		FB_ModbusRead_PowerCol		: ARRAY[1.. CstNbPowerCol_PCS_G] OF FB_ModbusRead;
		FB_ModbusRead_DU			: ARRAY[1..CstNb_DU_G] OF FB_ModbusRead;
		FB_ModbusRead	          	: ARRAY[1..6] OF FB_ModbusRead; // (NA) FB for Modbus Reading
		FB_ModbusWrite				: ARRAY[1..7]  OF FB_ModbusWrite;
		AX_ModbusReadAlarmPowerCol	: ARRAY[1.. CstNbPowerCol_PCS_G] OF BOOL;
		AX_ModbusReadAlarmDU		: ARRAY[1.. CstNb_DU_G] OF BOOL;
		AX_ModbusReadAlarm			: ARRAY[1..6] OF BOOL;
		AX_ModbusReadAlarmId		: ARRAY[1..11] OF UDINT;
		AX_ModbusReadAlarmIdPowerCol: ARRAY[1.. CstNbPowerCol_PCS_G] OF UDINT;	
		AX_ModbusReadAlarmId_DU		: ARRAY[1.. CstNb_DU_G] OF UDINT;	
		AX_ModbusWriteAlarm			: ARRAY[1..7]  OF BOOL;
		AX_ModbusWriteAlarmId		: ARRAY[1..7]  OF UDINT;	
	
		MesBlock_Temp_1 			: ARRAY [1..120] OF WORD ; 		// (NA) Temporary Block with multiple modbus reading 
		MesBlock_Temp_2 			: ARRAY [0..120] OF WORD ; 		// (NA) Temporary Block with multiple modbus reading 
		MesBlock_Temp_3 			: ARRAY [1..120] OF WORD ; 		// (NA) Temporary Block with multiple modbus reading 
		MesBlock_Temp_4 			: ARRAY [1..120] OF WORD ; 		// (NA) Temporary Block with multiple modbus reading 
		MesBlock_Temp_5 			: ARRAY[1..CstNbPowerCol_PCS_G] OF ARRAY [1..32] OF WORD; 	// (NA) Temporary Block with multiple modbus reading 
		MesBlock_Temp_6 			: ARRAY[1..CstNb_DU_G] OF ARRAY [1..6] OF WORD ; 				// (NA) Temporary Block with multiple modbus reading 
		MesBlockWrite1_Temp 		: WORD;							// (NA) Temporary Block with multiple modbus writing (Caution : Double Word variables)
		MesBlockWrite2_Temp			: ARRAY[1..3] OF WORD;			// (NA) Temporary Block with multiple modbus writing (Caution : Double Word variables)
		MesBlockWrite3_Temp			: WORD;							// (NA) Temporary Block with multiple modbus writing (Caution : Double Word variables)
		MesBlockWrite4_Temp			: ARRAY[1..10] OF WORD;			// (NA) Temporary Block with multiple modbus writing (Caution : Double Word variables)
		MesBlockWrite5_Temp			: ARRAY[1..2] OF WORD;
		MesBlockWrite6_Temp			: WORD;
		MesBlockWrite7_Temp			: ARRAY[1..2] OF WORD;
		MesBlockWrite8_Temp			: WORD;

		TON_BJ						: ARRAY[1..10] OF TON; 


		AX_ADR_MB_Write				: ARRAY[1..2] OF  WORD := [100, 557];		// [40553, 40558, 40551];
		AX_QTY_MB_Write				: ARRAY[1..2] OF  BYTE := [1, 	1];                    // [1, 1, 1];
		                    		
		InvSetptP_temp				: REAL;
		InvSetptQ_temp				: REAL;
                            		
                            		
		AX_QTY_MB					: ARRAY[1..8] OF WORD := [120, 	120, 	10, 	1, 		5, 		120, 	120, 	50];
		AX_ADR_MB					: ARRAY[1..8] OF WORD := [1000, 1119, 	550, 	1391, 	5000, 	0000, 	5803, 	1350]; 			
		
	// M_STARTSTOP//
		StartStop_RTrig				: R_Trig;
              	
	// M_CP
		CalCP_CMD_StartStop			: BOOL; 						// Write command start;
		
		bTestComAlarm : BOOL;
		bTestComWarning : BOOL;
END_VAR

METHOD M_AlarmManagement
//////////////////
// Manages IntelliGen Alarms
/////////////////

VAR 
	// Method local variables (reinitialized at each cycle) 
	FB_AlarmCodeManager : FB_AlarmCodeManager ; 
	KK				: BYTE;		// For Loop 
	bComError		: BOOL := TRUE;
	bComWarning 	: BOOL;

	AX_BJHS			: ARRAY[1..10] OF BOOL;
END_VAR

bComError := (AX_ModbusReadAlarmPowerCol[1] AND AX_ModbusReadAlarmPowerCol[2] AND AX_ModbusReadAlarmPowerCol[3] AND AX_ModbusReadAlarmPowerCol[4] AND AX_ModbusReadAlarmPowerCol[5] AND AX_ModbusReadAlarmPowerCol[6]
		AND AX_ModbusReadAlarm[1] AND AX_ModbusReadAlarm[2] AND AX_ModbusReadAlarm[3] AND AX_ModbusReadAlarm[4]
		AND AX_ModbusWriteAlarm[1] AND AX_ModbusWriteAlarm[2]) OR bTestComAlarm;

bComWarning:= AX_ModbusReadAlarmPowerCol[1] OR AX_ModbusReadAlarmPowerCol[2] OR AX_ModbusReadAlarmPowerCol[3] OR AX_ModbusReadAlarmPowerCol[4] OR AX_ModbusReadAlarmPowerCol[5] OR AX_ModbusReadAlarmPowerCol[6]
		OR AX_ModbusReadAlarm[1] OR AX_ModbusReadAlarm[2] OR AX_ModbusReadAlarm[3] OR AX_ModbusReadAlarm[4]
		OR AX_ModbusWriteAlarm[1] OR AX_ModbusWriteAlarm[2] or bTestComWarning;


TON_ComAlarm(IN := bComError, PT := T#30S,Q=> MesDataExd.MesData.MesAlarmCom);
TON_ComWarning(IN := bComWarning, PT := T#30S, Q=> MesWarningCom);

// ALARM CODE //
	FB_AlarmCodeManager(
		bAlarm1			:= NOT MesDataExd.MesStateCom,							// INV Not Communicating
		bAlarm2			:= FALSE,												// 	
		bAlarm3			:= NOT MesDataExd.MesStateCBac,							// INV AC CB opened 
		bAlarm4			:= FALSE,												// 	
		bAlarm5			:= NOT MesDataExd.MesStateCBdc,							// INV DC CB opened 
		bAlarm6			:= FALSE,												// 
		bAlarm7			:= MesDataExd.MesFaultGnd,								// INV Ground Fault	
		bAlarm8			:= FALSE,												// 
		bAlarm9			:= NOT MesDataExd.MesStateNoAlert, 						// INV ID = 9, inverter has detected an abnormal fault which prevents operation
		bAlarm10		:= FALSE, //
		bAlarm11		:= FALSE, //
		bAlarm12		:= FALSE, //
		bAlarm13		:= FALSE, //
		bAlarm14		:= FALSE, //
		bAlarm15		:= MesDataExd.MesData.MesAlarmCom, 						 // No communication frames for the past 30 seconds 					 			#COM
		wAlarmCode		=> MesDataExd.MesData.MesAlarmCode);					

// WARNING CODE //
	FB_AlarmCodeManager(
 		bAlarm1			:= MesWarningCom, 										// A frame failed for the last 30s 												#COM
		bAlarm2			:= FALSE, //
		bAlarm3			:= NOT MesDataExd.Mesdata.MesCP_Read, 	  							// No permission to read from SCADA
		bAlarm4			:= MesDataExd.ParamID_PMode <> 0,						// INV active power setpoint is not MPPT  										#Equipment
		bAlarm5			:= NOT MesDataExd.Mesdata.MesCP_Write,								// No permission to write from SCADA							
		bAlarm6			:= FALSE, //
		bAlarm7			:= FALSE, //
		bAlarm8			:= FALSE,												//
		bAlarm9			:= IN_SetptPlimit_Local < ParamPn,  	// INV local active power setpoint is under nominal active power 
		bAlarm10		:= NOT RS_StartStop_Local.Q1,       					// Local Stop Command 
		bAlarm11		:= FALSE,						 						// 
		bAlarm12		:= FALSE, 												//
		bAlarm13		:= FALSE,												// 
		bAlarm14		:= FALSE,												// 
		bAlarm15		:= FALSE, 												//
		wAlarmCode		=> MesDataExd.MesData.MesWarningCode);	
// EVENT CODE //
	FB_AlarmCodeManager(
		bAlarm1			:= FALSE, //
		bAlarm2			:= FALSE, //
		bAlarm3			:= FALSE, //
		bAlarm4			:= FALSE, //
		bAlarm5			:= FALSE, //
		bAlarm6			:= FALSE, //
		bAlarm7			:= MesDataExd.MesData.MesState_INV = 24,  				// Econmode: activated the econmode to save MV losses
		bAlarm8			:= MesDataExd.MesData.MesState_INV = 23,  				// Autonight: switches to autonight state
		bAlarm9			:= MesDataExd.MesData.MesState_INV = 20,  				// Premagnetization: MV transformer pre-mag
		bAlarm10		:= MesDataExd.MesData.MesState_INV = 19,  				// Filter contactors: LC filter contact activated
		bAlarm11		:= NOT RS_StartStop.Q1, 								// Stop command for INV 
		bAlarm12		:= MesDataExd.MesData.MesState_INV = 0,  				// Power Up
		bAlarm13		:= MesDataExd.MesData.MesState_INV = 1,  				// Init: basic condition are being checked
		bAlarm14		:= MesDataExd.MesData.MesState_INV = 2,  				// Off: stopped
		bAlarm15		:= MesDataExd.MesData.MesState_INV = 3,  				// PCHG : Precharge
		wAlarmCode		=>  MesDataExd.MesData.MesEventCode);
// EVENT CODE //
	FB_AlarmCodeManager(
		bAlarm1			:= MesDataExd.MesData.MesState_INV = 4,  				// REA : Ready, wainting for start command
		bAlarm2			:= MesDataExd.MesData.MesState_INV = 5,  				// WAIT: Waiting for delay time
		bAlarm3			:= MesDataExd.MesData.MesState_INV = 6,  				// ON: inverter operting normally
		bAlarm4			:= MesDataExd.MesData.MesState_INV = 7,  				// Stop: inverter is stopping
		bAlarm5			:= MesDataExd.MesData.MesState_INV = 8,  				// Discharge: capacitor discharging for 1min
		bAlarm6			:= MesDataExd.MesData.MesState_INV = 9,  				// Fault: check fault code
		bAlarm7			:= MesDataExd.MesData.MesState_INV = 10,  				// LVRT: low voltage ride through
		bAlarm8			:= MesDataExd.MesData.MesState_INV = 11,  				// OVRT: Over voltage ride through
		bAlarm9			:= MesDataExd.MesData.MesState_INV = 12,  				// NGHT: Night
		bAlarm10		:= MesDataExd.MesData.MesState_INV = 13,  				// NDCO: Night DC off: DC opened, no heating or night mode
		bAlarm11		:= MesDataExd.MesData.MesState_INV = 14,  				// Standby: waiting for conditions to perform softcharge
		bAlarm12		:= MesDataExd.MesData.MesState_INV = 15,  				// HVPL: high voltage phase lost
		bAlarm13		:= MesDataExd.MesData.MesState_INV = 16,  				// Trackers: trackers mode running
		bAlarm14		:= MesDataExd.MesData.MesState_INV = 17,  				// Pre-on: soft charge and synchronization
		bAlarm15		:= MesDataExd.MesData.MesState_INV = 18,  				// Diagnosis: extended self-diagnosis									
		wAlarmCode		=>  MesDataExd.MesEventCode2);

				
(*
	FB_AlarmCodeManager(
		bAlarm0			:= FALSE, 			// P Curtail -  no curtail
		bAlarm1			:= FALSE, 			// P Curtail -  Id : Current close loop
		bAlarm2			:= FALSE, 			// P Curtail -  P : Power close loop
		bAlarm3			:= FALSE, 			// P Curtail -  Vdc : voltage close loop
		bAlarm4			:= FALSE, 			// P Curtail -  HT
		bAlarm5			:= FALSE, 			// P Curtail -  STAT
		bAlarm6			:= FALSE, 			// P Curtail -  R
		bAlarm7			:= FALSE, 			// P Curtail -  Night : voltage dc night
		bAlarm8			:= FALSE, 			// 
		bAlarm9			:= FALSE, 			// 
		bAlarm10		:= FALSE, 			// 
		bAlarm11		:= FALSE,			// 
		bAlarm12		:= FALSE,			// 
		bAlarm13		:= FALSE,			// 
		bAlarm14		:= FALSE,			// 
		bAlarm15		:= FALSE,			// 		
		wAlarmCode		=>  MesDataExd.MesStatusCurtail_P);

	FB_AlarmCodeManager(
		bAlarm0			:= FALSE, 			// Q Curtail - CosPhi
		bAlarm1			:= FALSE, 			// Q Curtail - Iq : Current close loop
		bAlarm2			:= FALSE, 			// Q Curtail - Q : Power cose loop
		bAlarm3			:= FALSE, 			// Q Curtail - QV : QV Curve
		bAlarm4			:= FALSE, 			// Q Curtail - HT
		bAlarm5			:= FALSE, 			// Q Curtail - R
		bAlarm6			:= FALSE, 			// 
		bAlarm7			:= FALSE, 			// 
		bAlarm8			:= FALSE, 			// 
		bAlarm9			:= FALSE, 			// 
		bAlarm10		:= FALSE, 			// 
		bAlarm11		:= FALSE,			// 
		bAlarm12		:= FALSE,			// 
		bAlarm13		:= FALSE,			// 
		bAlarm14		:= FALSE,			// 
		bAlarm15		:= FALSE,			// 		
		wAlarmCode		=>  MesDataExd.MesStatusCurtail_Q);

	FB_AlarmCodeManager(
		bAlarm0			:= FALSE, 			// State - Stopped
		bAlarm1			:= FALSE, 			// State - MPPT
		bAlarm2			:= FALSE, 			// State - Sleeping
		bAlarm3			:= FALSE, 			// State - Starting
		bAlarm4			:= FALSE, 			// State - Throttled
		bAlarm5			:= FALSE, 			// State - Shutting Down
		bAlarm6			:= FALSE, 			// State - Fault
		bAlarm7			:= FALSE, 			// State - Standby
		bAlarm8			:= FALSE, 			// 
		bAlarm9			:= FALSE, 			// 
		bAlarm10		:= FALSE, 			// 
		bAlarm11		:= FALSE,			// 
		bAlarm12		:= FALSE,			// 
		bAlarm13		:= FALSE,			// 
		bAlarm14		:= FALSE,			// 
		bAlarm15		:= FALSE,			// 		
		wAlarmCode		=>  MesDataExd.MesData.MesState);		
		
		
*)				
FOR KK := 1 TO CstNbPowerCol_PCS_G DO
	FB_AlarmCodeManager(
		bAlarm1			:= MesDataExd.AX_PowerCol[KK].MesState_Inv = 22, 			// 22, Idle: Module waits 5s before starting
		bAlarm2			:= MesDataExd.AX_PowerCol[KK].MesState_Inv = 1, 			// 1, Stop: Module is stopped
		bAlarm3			:= MesDataExd.AX_PowerCol[KK].MesState_Inv = 2, 			// 2, Softcharge: Module performing softcharge
		bAlarm4			:= MesDataExd.AX_PowerCol[KK].MesState_Inv = 3, 			// 3, Ready: waiting for start command
		bAlarm5			:= MesDataExd.AX_PowerCol[KK].MesState_Inv = 4, 			// 4, LCL: LCL filter contact activated
		bAlarm6			:= MesDataExd.AX_PowerCol[KK].MesState_Inv = 5, 			// 5, Main AC: main contact activated, waiting feedback
		bAlarm7			:= MesDataExd.AX_PowerCol[KK].MesState_Inv = 6, 			// 6, Main AC Wait: module waits 100ms with ac contact closed
		bAlarm8			:= MesDataExd.AX_PowerCol[KK].MesState_Inv = 7, 			// 7, Run: Module injecting
		bAlarm9			:= MesDataExd.AX_PowerCol[KK].MesState_Inv = 8, 			// 8, nMain AC: AC open, LCL contactor closed during 100ms
		bAlarm10		:= MesDataExd.AX_PowerCol[KK].MesState_Inv = 9, 			// 9, Discharge: Module performing active discharge
		bAlarm11		:= MesDataExd.AX_PowerCol[KK].MesState_Inv = 10,			// 10, VRT event occured in network
		bAlarm12		:= MesDataExd.AX_PowerCol[KK].MesState_Inv = 11,			// 11, Trackers mode
		bAlarm13		:= MesDataExd.AX_PowerCol[KK].MesState_Inv = 14,			// 14, Fault AC overcurrent
		bAlarm14		:= MesDataExd.AX_PowerCol[KK].MesState_Inv = 15,			// 15, Fault overvoltage
		bAlarm15		:= MesDataExd.AX_PowerCol[KK].MesState_Inv = 17,			// 17, Fault exit OV wait
		wAlarmCode		=>  MesDataExd.AX_PowerCol[KK].MesState_Inv_ID);	
		
		
	FB_AlarmCodeManager(
		bAlarm1			:= MesDataExd.AX_PowerCol[KK].MesState_Inv = 55, 			// 55,  Init : Module is initializing
		bAlarm2			:= MesDataExd.AX_PowerCol[KK].MesState_Inv = 18, 			// 18, Fault exit wait
		bAlarm3			:= MesDataExd.AX_PowerCol[KK].MesState_Inv = 19, 			// 19, Softcharge fault
		bAlarm4			:= MesDataExd.AX_PowerCol[KK].MesState_Inv = 20, 			// 20, Fault
		bAlarm5			:= MesDataExd.AX_PowerCol[KK].MesState_Inv = 116, 			// 116, Module disabled SC: softcharge fault
		bAlarm6			:= MesDataExd.AX_PowerCol[KK].MesState_Inv = 159, 			// 159, Master FPGA comms error
		bAlarm7			:= FALSE, //
		bAlarm8			:= FALSE, //
		bAlarm9			:= FALSE, //
		bAlarm10		:= FALSE, //
		bAlarm11		:= FALSE, //
		bAlarm12		:= FALSE, //
		bAlarm13		:= FALSE, //
		bAlarm14		:= FALSE, //
		bAlarm15		:= FALSE, //
		wAlarmCode		=>  MesDataExd.AX_PowerCol[KK].MesState_Inv_ID2);	
END_FOR
END_METHOD

METHOD M_CP
//////////////////
//  Emulator
/////////////////

VAR 
	// Method local variables (reinitialized at each cycle) 
	
END_VAR

	
SUPER^.M_CP();
CalCP_CMD_StartStop	:= FB_ModbusRead[1].OUT_NbRead > 0 AND SEL(MesDataExd.MesStartDisabled, TRUE, NOT RS_StartStop.Q1); // FB_ModbusRead[1].OUT_NbRead > 0 AND (MesDataExd.MesStartDisabled  <> NOT  RS_StartStop.Q1);  




Trig_Cmd_Read(CLK:=IN_CmdToggleRead);
Trig_Cmd_Write(CLK:=IN_CmdToggleWrite);
	
IF Trig_Cmd_Read.Q THEN
	IN_CmdToggleRead := FALSE;
	MesDataExd.MesData.MesCP_Read := NOT MesDataExd.MesData.MesCP_Read;
END_IF


IF Trig_Cmd_Write.Q THEN
	IN_CmdToggleWrite := FALSE;
	MesDataExd.MesData.MesCP_Write := NOT MesDataExd.MesData.MesCP_Write;
END_IF
END_METHOD

{attribute 'object_name' := 'M_Curtail'}
METHOD M_Curtail
//////////////////
// Write Curtail Command through modbus to PV inverters.  
//////////////////
VAR 
	// Method local variables (reinitialized at each cycle) 

	MW					: FB_MergeWordsToFloat;
	MW_1				: FB_SplitFloatToWords;

	KK: INT;
END_VAR
SUPER^.M_Curtail() ; 

// MODBUS VARIABLE FORMATING //
// Setpoints //

IF IN_SetptPlimit = 0 AND (MesDataExd.MesData.MesState.0 OR MesDataExd.MesData.MesState.2 OR MesDataExd.MesData.MesState.3) THEN
	IN_SetptPlimit := 100;
END_IF

IF MesDataExd.OUT_CmdInvLocal THEN
	InvSetptP_temp	:= 100*MIN(100, 100 * IN_SetptPlimit_Local / ParamPn); 
	InvSetptQ_temp	:= 100*MIN(100, 100 * IN_SetptQ_Local / ParamQn); 

	MesDataExd.MesData.OUT_SetptPLimit :=  IN_SetptPlimit_Local; 
	MesDataExd.MesData.OUT_SetptQ :=  IN_SetptQ_Local; 	

ELSE
	InvSetptP_temp	:= 10000*IN_SetptPlimit / ParamPn; 
	InvSetptQ_temp	:= 10000*IN_SetptQ / ParamQn; 

	MesDataExd.MesData.OUT_SetptPLimit :=  IN_SetptPlimit; 
	MesDataExd.MesData.OUT_SetptQ :=  IN_SetptQ; 
	
END_IF	

		
	
	MesBlockWrite4_Temp[1] := REAL_TO_WORD(InvSetptP_temp);
	MesBlockWrite4_Temp[2] := REAL_TO_WORD(InvSetptQ_temp);
			
		
		FB_ModbusWrite[1]
	(
		pSrcAddr := ADR (MesBlockWrite4_Temp[1]),
		sIPAddr := ParamIPAddress,
		tTimeout := ParamTimeout,
		nMBAddr := AX_ADR_MB_Write[1],
		nTCPport := ParamTCPPort,
		cbLength := SIZEOF(MesBlockWrite4_Temp[1]),
		nQuantity := AX_QTY_MB_Write[1],
		nUnitID := ParamUnitID,
		WriteCmd := ClockWrite AND MesDataExd.Mesdata.MesCP_Write  ,
		Reset := CmdClearFault_G OR IN_CmdReset_L,
		ErrorId => AX_ModbusWriteAlarmId[1],
		ModbusWriteAlarm => AX_ModbusWriteAlarm[1]
	);

	FB_ModbusWrite[2]
(
	pSrcAddr := ADR (MesBlockWrite4_Temp[2]),
	sIPAddr := ParamIPAddress,
	tTimeout := ParamTimeout,
	nMBAddr := AX_ADR_MB_Write[2],
	nTCPport := ParamTCPPort,
	cbLength := SIZEOF(MesBlockWrite4_Temp[2]),
	nQuantity := AX_QTY_MB_Write[2],
	nUnitID := ParamUnitID,
	WriteCmd := ClockWrite AND MesDataExd.Mesdata.MesCP_Write  ,
	Reset := CmdClearFault_G OR IN_CmdReset_L,
	ErrorId => AX_ModbusWriteAlarmId[2],
	ModbusWriteAlarm => AX_ModbusWriteAlarm[2]
);
END_METHOD

METHOD M_Evaluate
VAR_INPUT
END_VAR
IN_SetptPlimit 	:= IN_SetptPlimit;
IN_SetptQ		:= IN_SetptQ;
END_METHOD

METHOD M_Execute
//////////////////
//  Method Calls 
/////////////////

VAR 
	// Method local variables (reinitialized at each cycle) 

END_VAR
IF  bInit THEN
	M_Init();
	bInit:= FALSE ; 
ELSIF CmdInit_G THEN 
	bInit:= TRUE ;
END_IF

SUPER^.M_Execute(); 

//M_Evaluate();
M_AlarmManagement();
END_METHOD

METHOD M_Init

VAR
	bCompleted 			: BOOL := FALSE;
	AX_ADR_MB			: WORD := 44253; 
END_VAR
ParamPn := 3800;
IN_SetptPlimit_Local := 3800;

// Watchdog timer start
Watchdog_CP_Write := TRUE;
ParamClockReadTime := T#1S;
ParamClockWriteTime := T#200MS;
END_METHOD

{attribute 'object_name' := 'M_Read'}
METHOD M_Read
//////////
// Read Method for PE SKID HEMK : Modbus reading
//////////
VAR
	// Method local variables (reinitialized at each cycle) 
	MW_Float			: FB_MergeWordsToFloat;
	MW_REAL				: FB_MergeWordsToDint;
	MW_UInt				: FB_MergeWordsToUint;
	
	
	EacInj_Interm1		: ULINT;
	EacCon_Interm1		: ULINT;
	EreacCapa_Interm1	: ULINT;
	EreacInd_Interm1	: ULINT;
	EacInj_Day_Interm1	: ULINT;
	
	EacInj_Interm2		: ULINT;
	EacCon_Interm2		: ULINT;
	EreacCapa_Interm2	: ULINT;
	EreacInd_Interm2	: ULINT;
	EacInj_Day_Interm2	: ULINT;
	
	Temp_Cells_Transfo	: WORD;
	Temp_Cells_Transfo_2: WORD;
	Temp_Cells_Transfo_3: WORD;
	Temp_Cells_Transfo_4: WORD;
	MesResistor			: REAL;
	
	KK					: BYTE;						 // Index to loop over modbus blocks 	
	JJ					: BYTE;
END_VAR
IF MesDataExd.MesData.MesCP_Read THEN		

// MODBUS REQUEST//
	//Electrical Measurements + Ground Measurements
	FB_ModbusRead[1]
	(
		nTCPPort		:= ParamTcpPort,
		ClockRead		:= MesDataExd.Mesdata.MesCP_Read AND ClockRead, 
		Reset			:= CmdClearFault_G OR IN_CmdReset_L,
		sIPAddr			:=ParamIPAddress ,
		nUnitID			:= 1, 
		tTimeout		:= ParamTimeout,
		nQuantity		:= AX_QTY_MB[1] , 
		nMBAddr			:= AX_ADR_MB[1] , 
		cbLength		:= SIZEOF(MesBlock_Temp_1) , 
		pDestAddr		:= ADR(MesBlock_Temp_1) , 
		ModbusReadAlarm	=>AX_ModbusReadAlarm[1] , 
		ErrorId			=> AX_ModbusReadAlarmId[1]
	);
		
	//Production Measurements
	FB_ModbusRead[2]
	(
		nTCPPort		:= ParamTcpPort,
		ClockRead		:= MesDataExd.Mesdata.MesCP_Read AND ClockRead, 
		Reset			:= CmdClearFault_G OR IN_CmdReset_L,
		sIPAddr			:=ParamIPAddress , 
		nUnitID			:= 1, 
		tTimeout		:= ParamTimeout,
		nQuantity		:= AX_QTY_MB[2] , 
		nMBAddr			:= AX_ADR_MB[2] , 
		cbLength		:= SIZEOF(MesBlock_Temp_2) , 
		pDestAddr		:= ADR(MesBlock_Temp_2) , 
		ModbusReadAlarm	=>AX_ModbusReadAlarm[2] , 
		ErrorId			=> AX_ModbusReadAlarmId[2]
	);
	
	// Status Summary + Event Summary
	FB_ModbusRead[3]
	(
		nTCPPort		:= ParamTcpPort,
		ClockRead		:= MesDataExd.MesData.MesCP_Read AND ClockRead, 
		Reset			:= CmdClearFault_G OR IN_CmdReset_L,
		sIPAddr			:=ParamIPAddress , 
		nUnitID			:= 1, 
		tTimeout		:= ParamTimeout,
		nQuantity		:= AX_QTY_MB[3] , 
		nMBAddr			:= AX_ADR_MB[3] , 
		cbLength		:= SIZEOF(MesBlock_Temp_3) , 
		pDestAddr		:= ADR(MesBlock_Temp_3) , 
		ModbusReadAlarm	=>AX_ModbusReadAlarm[3] , 
		ErrorId			=> AX_ModbusReadAlarmId[3]
	);
	
	//Number running modules
	FB_ModbusRead[4]
	(
		nTCPPort		:= ParamTcpPort,
		ClockRead		:= MesDataExd.MesData.MesCP_Read AND ClockRead, 
		Reset			:= CmdClearFault_G OR IN_CmdReset_L,
		sIPAddr			:= ParamIPAddress , 
		nUnitID			:= 1, 
		tTimeout		:= ParamTimeout,
		nQuantity		:= AX_QTY_MB[4], 
		nMBAddr			:= AX_ADR_MB[4], 
		cbLength		:= SIZEOF(MesBlock_Temp_4), 
		pDestAddr		:= ADR(MesBlock_Temp_4), 
		ModbusReadAlarm	=> AX_ModbusReadAlarm[4], 
		ErrorId			=> AX_ModbusReadAlarmId[4]
	);
	
	//Power Commands
	FOR KK:= 1 TO  CstNbPowerCol_PCS_G DO 
		FB_ModbusRead_PowerCol[KK]
		(
				nTCPPort		:= ParamTcpPort,
				ClockRead		:= MesDataExd.Mesdata.MesCP_Read AND ClockRead, 
				Reset			:= CmdClearFault_G OR IN_CmdReset_L,
				sIPAddr			:=ParamIPAddress , 
				nUnitID			:= 1, 
				tTimeout		:= ParamTimeout,
				nQuantity		:= 32 , 
				nMBAddr			:= 5000 + 32*(KK-1) ,  
				cbLength		:= SIZEOF(MesBlock_Temp_5[KK]) , 
				pDestAddr		:= ADR(MesBlock_Temp_5[KK]) , 
				ModbusReadAlarm	=>AX_ModbusReadAlarmPowerCol[KK] , 
				ErrorId			=> AX_ModbusReadAlarmIdPowerCol[KK]
		);
	END_FOR
		
	FOR KK:= 1 TO  CstNb_DU_G DO 
		FB_ModbusRead_DU[KK]
		(
				nTCPPort		:= ParamTcpPort,
				ClockRead		:= MesDataExd.Mesdata.MesCP_Read AND ClockRead, 
				Reset			:= CmdClearFault_G OR IN_CmdReset_L,
				sIPAddr			:= ParamIPAddress , 
				nUnitID			:= 1, 
				tTimeout		:= ParamTimeout,
				nQuantity		:= 6, 
				nMBAddr			:= 5800 + 6*(KK-1),  
				cbLength		:= SIZEOF(MesBlock_Temp_6[KK]), 
				pDestAddr		:= ADR(MesBlock_Temp_6[KK]), 
				ModbusReadAlarm	=>AX_ModbusReadAlarmDU[KK], 
				ErrorId			=> AX_ModbusReadAlarmId_DU[KK]
		);
	END_FOR
      

    MW_REAL(WORD_STRONG:= MesBlock_Temp_1[  1], SIGNED:=FALSE, FIX:=0 , SIZE:=1, VAR_OUT:=MesDataExd.MesU12);
	MW_REAL(WORD_STRONG:= MesBlock_Temp_1[  2], SIGNED:=FALSE, FIX:=0 , SIZE:=1, VAR_OUT:=MesDataExd.MesU23);
	MW_REAL(WORD_STRONG:= MesBlock_Temp_1[  3], SIGNED:=FALSE, FIX:=0 , SIZE:=1, VAR_OUT:=MesDataExd.MesU31);
	MW_REAL(WORD_STRONG:= MesBlock_Temp_1[  4], SIGNED:=FALSE, FIX:=1 , SIZE:=1, VAR_OUT:=MesDataExd.MesI1);
	MW_REAL(WORD_STRONG:= MesBlock_Temp_1[  5], SIGNED:=FALSE, FIX:=1 , SIZE:=1, VAR_OUT:=MesDataExd.MesI2);
	MW_REAL(WORD_STRONG:= MesBlock_Temp_1[  6], SIGNED:=FALSE, FIX:=1 , SIZE:=1, VAR_OUT:=MesDataExd.MesI3);
	MW_REAL(WORD_STRONG:= MesBlock_Temp_1[  8], SIGNED:=TRUE, FIX:=0 , SIZE:=1, VAR_OUT:=MesDataExd.MesData.MesP);
	MW_REAL(WORD_STRONG:= MesBlock_Temp_1[  9], SIGNED:=TRUE, FIX:=0 , SIZE:=1, VAR_OUT:=MesDataExd.MesData.MesQ);
	MW_REAL(WORD_STRONG:= MesBlock_Temp_1[ 10], SIGNED:=FALSE, FIX:=0 , SIZE:=1, VAR_OUT:=MesDataExd.MesData.MesS);
	MW_REAL(WORD_STRONG:= MesBlock_Temp_1[ 11], SIGNED:=TRUE, FIX:=3 , SIZE:=1, VAR_OUT:=MesDataExd.MesData.MesCosPhi);
	MW_REAL(WORD_STRONG:= MesBlock_Temp_1[ 12], SIGNED:=FALSE, FIX:=2 , SIZE:=1, VAR_OUT:=MesDataExd.MesData.MesFreq);
	MW_REAL(WORD_STRONG:= MesBlock_Temp_1[ 52], SIGNED:=FALSE, FIX:=0 , SIZE:=1, VAR_OUT:=MesDataExd.MesData.MesUdc);  
	MW_REAL(WORD_STRONG:= MesBlock_Temp_1[ 61], SIGNED:=FALSE, FIX:=0 , SIZE:=1, VAR_OUT:=MesDataExd.MesData.MesPdc);
	MW_REAL(WORD_STRONG:= MesBlock_Temp_1[ 62], SIGNED:=FALSE, FIX:=0 , SIZE:=1, VAR_OUT:=MesDataExd.MesData.MesIdc); 
	MW_REAL(WORD_STRONG:= MesBlock_Temp_1[ 104], Word_WEAK:= MesBlock_Temp_1[105], SIGNED:=FALSE, FIX:=3 , SIZE:=2, VAR_OUT:=MesDataExd.MesData.MesInsuResistor);
	MW_REAL(WORD_STRONG:= MesBlock_Temp_1[ 114], Word_WEAK:= MesBlock_Temp_1[115], SIGNED:=FALSE, FIX:=0 , SIZE:=2, VAR_OUT:=MesDataExd.MesInsuResistor_AC);
	

	
	
// INV status
	MW_REAL(WORD_STRONG:= MesBlock_Temp_2[ 0], SIGNED:=FALSE, FIX:=0 , SIZE:=1, VAR_OUT:=MesDataExd.MesTemp_DU);
	MW_UInt(WORD_STRONG:= MesBlock_Temp_2[ 1], VAR_OUT := MesDataExd.MesAlarm_Control); 	
	MW_UInt(WORD_STRONG:= MesBlock_Temp_2[ 2], VAR_OUT := MesDataExd.MesWarning_Control); 	
	MW_UInt(WORD_STRONG:= MesBlock_Temp_2[ 3], VAR_OUT := MesDataExd.MesData.MesState_INV); 	
	MW_REAL(WORD_STRONG:= MesBlock_Temp_2[ 4], SIGNED:=FALSE, FIX:=0 , SIZE:=1, VAR_OUT:=MesDataExd.MesTemp_Control);
	MW_REAL(WORD_STRONG:= MesBlock_Temp_2[ 5], SIGNED:=FALSE, FIX:=0 , SIZE:=1, VAR_OUT:=MesDataExd.MesTemp_IGBTmax);
	MW_REAL(WORD_STRONG:= MesBlock_Temp_2[ 6], SIGNED:=FALSE, FIX:=0 , SIZE:=1, VAR_OUT:=MesDataExd.MesTemp_PowerColmax);	

	MW_REAL(WORD_STRONG:= MesBlock_Temp_2[21], SIGNED:=FALSE, FIX:=4, SIZE:=1, VAR_OUT:=MesDataExd.MesSetptP);
	MW_REAL(WORD_STRONG:= MesBlock_Temp_2[22], SIGNED:=FALSE, FIX:=4, SIZE:=1, VAR_OUT:=MesDataExd.MesSetptQ);
	MesDataExd.MesCP_Start := WORD_TO_BOOL(MesBlock_Temp_2[ 31]);
	
// Power column/module variables
		MesDataExd.MesStatusCurtail_P := MesBlock_Temp_3[1]; 
		MesDataExd.MesStatusCurtail_Q := MesBlock_Temp_3[2]; 

	
		MesDataExd.MesNbRunningModules := WORD_TO_UINT(MesBlock_Temp_4[1]);
	
	FOR KK:= 1 TO CstNbPowerCol_PCS_G DO 	
		MW_UInt(WORD_STRONG:= MesBlock_Temp_5[KK][ 1], VAR_OUT := MesDataExd.AX_PowerCol[KK].MesState_Inv);
	
		MW_REAL(WORD_STRONG:= MesBlock_Temp_5[KK][ 2], SIGNED:=FALSE, FIX:=1 , SIZE:=1, VAR_OUT := MesDataExd.AX_PowerCol[KK].MesData.MesI1);
		MW_REAL(WORD_STRONG:= MesBlock_Temp_5[KK][ 3], SIGNED:=FALSE, FIX:=1 , SIZE:=1, VAR_OUT := MesDataExd.AX_PowerCol[KK].MesData.MesI2);
		MW_REAL(WORD_STRONG:= MesBlock_Temp_5[KK][ 4], SIGNED:=FALSE, FIX:=1 , SIZE:=1, VAR_OUT := MesDataExd.AX_PowerCol[KK].MesData.MesI3);
		MW_REAL(WORD_STRONG:= MesBlock_Temp_5[KK][ 5], SIGNED:=FALSE, FIX:=1 , SIZE:=1, VAR_OUT := MesDataExd.AX_PowerCol[KK].MesData.MesIdc);
		MW_REAL(WORD_STRONG:= MesBlock_Temp_5[KK][ 8], SIGNED:=FALSE, FIX:=0 , SIZE:=1, VAR_OUT := MesDataExd.AX_PowerCol[KK].MesData.MesUdc);
		MW_REAL(WORD_STRONG:= MesBlock_Temp_5[KK][ 9], SIGNED:=FALSE, FIX:=1 , SIZE:=1, VAR_OUT := MesDataExd.AX_PowerCol[KK].MesData.MesP);
		MW_REAL(WORD_STRONG:= MesBlock_Temp_5[KK][ 10], SIGNED:=FALSE, FIX:=1 , SIZE:=1, VAR_OUT:= MesDataExd.AX_PowerCol[KK].MesData.MesQ);
		MW_REAL(WORD_STRONG:= MesBlock_Temp_5[KK][ 11], SIGNED:=FALSE, FIX:=0 , SIZE:=1, VAR_OUT:= MesDataExd.AX_PowerCol[KK].MesTemp);
		MW_REAL(WORD_STRONG:= MesBlock_Temp_5[KK][ 12], SIGNED:=FALSE, FIX:=0 , SIZE:=1, VAR_OUT:= MesDataExd.AX_PowerCol[KK].MesTempmax);
		
		MesDataExd.AX_PowerCol[KK].MesStateIO := MesBlock_Temp_5[KK][13];
		MW_REAL(WORD_STRONG:= MesBlock_Temp_5[KK][ 32], SIGNED:=FALSE, FIX:=0 , SIZE:=1, VAR_OUT:=MesDataExd.AX_PowerCol[KK].MesHygro);
	END_FOR
		
	//// DU Channels ///////
	FOR KK:= 1 TO CstNb_DU_G DO 
	// Status
		MW_UInt(WORD_STRONG:= MesBlock_Temp_6[KK][4], VAR_OUT := MesDataExd.AX_DU[KK].MesIDState); 
			
	// Current
		MW_REAL(WORD_STRONG:= MesBlock_Temp_6[KK][5], SIGNED:=TRUE, FIX:=1, SIZE:=1, VAR_OUT := MesDataExd.AX_DU[KK].MesI); // dA ?
	
	// Voltage
		MW_REAL(WORD_STRONG:= MesBlock_Temp_6[kk][6], SIGNED:=TRUE, FIX:=1, SIZE:=1, VAR_OUT := MesDataExd.AX_DU[KK].MesU); // dV ?
				
	END_FOR
	// Evaluate 
	MesDataExd.MesData.MesI						:= (MesDataExd.MesI1 + MesDataExd.MesI2 + MesDataExd.MesI3) /3;
	MesDataExd.MesData.MesU						:= (MesDataExd.MesU12 + MesDataExd.MesU23 + MesdataExd.MesU31) /3 ; 
	                                			
	MesDataExd.MesData.MesAlarmCom  			:= TON_ComAlarm.Q; 
	MesDataExd.MesStateCom 						:= NOT MesDataExd.MesData.MesAlarmCom; 
	MesDataExd.MesData.MesTemp					:= MesDataExd.MesTemp_Control;                         			                                    	
END_IF
END_METHOD

METHOD M_StartStop
VAR
	KK : UINT;
	AX_ADR_MB			: ARRAY[1..3] OF WORD := [43010, 43200, 44252];
	AX_QTY_MB			: ARRAY[1..3] OF BYTE := [3, 1, 1];
END_VAR
SUPER^.M_StartStop(); 

// Start/Stop
Trig_Local_Start(CLK:=IN_CmdStart_Local);
Trig_Local_Stop(CLK:=IN_CmdStop_Local);

Trig_Start(CLK:=IN_CmdStart);
Trig_Stop(CLK:=IN_CmdStop);

IF Trig_Local_Start.Q OR Trig_Local_Stop.Q OR Trig_Stop.Q OR Trig_Start.Q THEN
	RS_StartStop(SET:=(IN_CmdStart_Local AND NOT IN_CmdStop_Local) OR (IN_CmdStart AND NOT (IN_CmdStop OR IN_CmdStop_Local)), 
			 Reset1 := IN_CmdStop_Local OR (IN_CmdStop AND NOT IN_CmdStart_Local)); 
END_IF

// Emergency stop 
Trig_Local_EmergencyStop(CLK:=IN_CmdEmergencyStop_Local);

// Reset 
Trig_Reset(CLK:= IN_CmdReset_L);

FB_ModbusWrite[5](WriteCmd := FALSE);
FB_ModbusWrite[6](WriteCmd := FALSE);
//FB_ModbusWrite[7](WriteCmd := FALSE);

// Start/Stop/Reset
MesBlockWrite2_Temp[1] := BOOL_TO_WORD(RS_StartStop.Q1);
MesBlockWrite2_Temp[2] := BOOL_TO_WORD(NOT RS_StartStop.Q1);
MesBlockWrite2_Temp[3] := BOOL_TO_WORD(Trig_Reset.Q);
// Emergency stop 
MesBlockWrite3_Temp    := BOOL_TO_WORD(Trig_Local_EmergencyStop.Q);

MesDataExd.MesData.OUT_CmdStart := RS_StartStop.Q1 ; 
MesDataExd.MesData.OUT_CmdStop  := NOT RS_StartStop.Q1 ; 	
MesDataExd.OUT_CmdReset			:= 	Trig_Reset.Q;
MesDataExd.OUT_CmdEmergencyStop := Trig_Local_EmergencyStop.Q;

StartStop_RTrig(CLK:=CalCP_CMD_StartStop);

	FB_ModbusWrite[5]
	(
		pSrcAddr := ADR (MesBlockWrite2_Temp),
		sIPAddr := ParamIPAddress,
		tTimeout := ParamTimeout,
		nMBAddr := AX_ADR_MB[1],
		nTCPport := ParamTCPPort,
		cbLength := SIZEOF(MesBlockWrite2_Temp),
		nQuantity := AX_QTY_MB[1],
		nUnitID := ParamUnitID,
		WriteCmd := StartStop_RTrig.Q AND MesDataExd.Mesdata.MesCP_Write ,
		Reset := CmdClearFault_G,
		ErrorId => AX_ModbusWriteAlarmId[5],
		ModbusWriteAlarm => AX_ModbusWriteAlarm[5]
	);

	FB_ModbusWrite[6]
	(
		pSrcAddr := ADR (MesBlockWrite3_Temp),
		sIPAddr := ParamIPAddress,
		tTimeout := ParamTimeout,
		nMBAddr := AX_ADR_MB[2],
		nTCPport := ParamTCPPort,
		cbLength := SIZEOF(MesBlockWrite3_Temp),
		nQuantity := AX_QTY_MB[2],
		nUnitID := ParamUnitID,
		WriteCmd := Trig_Local_EmergencyStop.Q AND MesDataExd.Mesdata.MesCP_Write,
		Reset := CmdClearFault_G,
		ErrorId => AX_ModbusWriteAlarmId[6],
		ModbusWriteAlarm => AX_ModbusWriteAlarm[6]
	);

// INV watchdog timer: for the first version of the code, this feature is not used and the watchdog is turned timer off. Developped for future uses.
// Write register every second 
//TP_Watchdog(IN:= Watchdog_CP_Write, PT:=TIME#1S);
//FTrig_Watchdog(CLK:=TP_Watchdog.Q);
//Watchdog_CP_Write := FTrig_Watchdog.Q;
//
//MesBlockWrite8_Temp := INT_TO_WORD(1);
//
//	FB_ModbusWrite[7]
//(
//	pSrcAddr  := ADR (MesBlockWrite8_Temp),
//	sIPAddr   := ParamIPAddress,
//	tTimeout  := ParamTimeout,
//	nMBAddr   := AX_ADR_MB[3],
//	nTCPport  := ParamTCPPort,
//	cbLength  := SIZEOF(MesBlockWrite8_Temp),
//	nQuantity := AX_QTY_MB[3],
//	nUnitID   := ParamUnitID,
//	WriteCmd  := MesData.MesCP_Write AND Watchdog_CP_Write,
//	Reset     := CmdClearFault_G,
//	ErrorId => AX_ModbusWriteAlarmId[7],
//	ModbusWriteAlarm => AX_ModbusWriteAlarm[7]
//);
//
END_METHOD

METHOD M_StateManager
//////////////////
// Detect which is the state of the inverter. IF loss of communication MesState =0, the last inverter state is kept  
/////////////////

VAR 
	// Method local variables (reinitialized at each cycle) 

	
END_VAR
//MesState_INV : HEMK
// 0 = Power Up	, 3 = Standby DC	, 6 = Ready DC	, 9 = Ready		, 12 = ON		, 15 = Diagnostic AC	
// 1 = Init 	, 4 = Precharge DC	, 7 = Standby AC, 10 = Wait 	, 13 = Stop 	, 16 = Discharge 		 			  		
// 2 = OFF		, 5 = Softcharge DC	, 8 = Blackstart, 11 = Pre ON	, 14 = Ready AC , 17 = Fault

// HEMS / HEMG
// 0 = Power Up>3	, 3 = Precharge>3	, 		6 = ON>1, 		9 = Fault>6,		12 = Night>7, 			15 = High Voltage Phase Lost>6,		18 = Diagnosis>3				23 = AutoNight>7
// 1 = Init >3	, 4 = Ready>7, 			7 = Stop>0, 		10 = LVRT>4, 		13 = Night dc off>0,		16 = Trackers>3 		 			  	19 = Filter contactors>3		24 = Econmode>7
// 2 = OFF>0		, 5 = Wait>3, 			8 = Discharge>5, 	11 = OVRT>4, 		14 = Standby>7,			17 = Pre-On>3							20 = Premagnetization>3

//MesState
//0=Stopped, 1 = MPPT, 2 = Sleeping, 3 = Starting, 4 = Throttled, 5 = Shutting down, 6 = Fault, 7 = Standby

MesDataExd.MesData.MesState := 0; 


IF MesDataExd.MesData.MesState_INV = 7 OR MesDataExd.MesData.MesState_INV = 2 OR MesDataExd.MesData.MesState_INV = 13 THEN
	MesDataExd.MesData.MesState.0 := 1; // Off

ELSIF MesDataExd.MesData.MesState_INV = 6  AND MesDataExd.MesStatusCurtail_P = 0 THEN
	MesDataExd.MesData.MesState.1 := 1; // MPPT
	
ELSIF 	MesDataExd.MesData.MesState_INV = 0 OR MesDataExd.MesData.MesState_INV = 1 OR MesDataExd.MesData.MesState_INV = 3  OR 
		MesDataExd.MesData.MesState_INV = 5 OR MesDataExd.MesData.MesState_INV = 16 OR MesDataExd.MesData.MesState_INV = 17  OR MesDataExd.MesData.MesState_INV = 18
	OR MesDataExd.MesData.MesState_INV = 19 OR MesDataExd.MesData.MesState_INV = 20 THEN
	MesDataExd.MesData.MesState.3 := 1; // Starting 
	
ELSIF MesDataExd.MesData.MesState_INV = 6 AND MesDataExd.MesStatusCurtail_P = 2 THEN
	MesDataExd.MesData.MesState.4 := 1; // Curtaling 

ELSIF MesDataExd.MesData.MesState_INV = 8 THEN
	MesDataExd.MesData.MesState.5 := 1; // Shutdown
 
ELSIF MesDataExd.MesData.MesState_INV = 9 OR MesDataExd.MesData.MesState_INV = 15  THEN
	MesDataExd.MesData.MesState.6 := 1; // Fault 
	
ELSE
	MesDataExd.MesData.MesState.7 := 1;  // Standby 
	
END_IF



SUPER^.M_StateManager();
END_METHOD

END_FUNCTION_BLOCK

// ---- 04_Application/ALARM/FUN_Alarms.TcPOU
PROGRAM FUN_Alarms
VAR_INPUT
	IN_Directory					: STRING := 'C:\Users\Administrator\Documents\Historisation\';	// Directory where the alarms are saved in csv
	ParamDisableSMS					: BOOL ;	// True : SMS Serveur is disabled 
	AX_MesAlarmCode				: ARRAY [0..CstNbAlarmCode] OF WORD;    // Tableau de Word avec tous les AlarmCode 

	
	ParamDelayForceAlarm : TIME := T#2S ; 
	bTriggerCount	: BOOL;
	nCountSequence	: INT := 1;
	bTestForceAlarms 	: BOOL;
	MesAlarmWordTestJulienDecouple	: ARRAY[1..CstNbAlarmCode+1] OF WORD;
		
END_VAR

VAR_INPUT PERSISTENT
	AX_Journal						: ARRAY [0..CstNbAlarmCode] OF ARRAY[0..15] OF ST_ValuesAlarms; //Journal d'envoi, contient destinataire et message, et gestion de l'envois ou pas du sms
	bFactoryReset					: BOOL:= TRUE ;
END_VAR



VAR
	AX_RecupWord 					: ARRAY [0..CstNbAlarmCode] OF WORD;

	
	// M_ALARMPROCESSING	



		
	//	FB_Flicker					: ARRAY [0..CstNbAlarmCode] OF ARRAY[0..15] OF FB_DetectFlicker ; 
		
	// CSV

	
	//MAIL

	//SMS
	


	TON_TriggerCount	: TON;
	F_TRIG_TriggerCount	: F_TRIG;

	
END_VAR

IF bFactoryReset THEN
	M_Init();
	///////// 
END_IF

M_AlarmManager();
M_AlarmProcessing();
	
// Ici, on prend surtout en compte les alarmes 
FUN_Alarms_CSV(ParamSeparateur := ';',ParamExtension := '.csv');

IF MAIN.OUT_CalRunningPLC_IO THEN
	FUN_SendMail();
	SMS_Server (IN_AX_Journal := AX_Journal);
	InfluxDb_AlarmsManagement() ; 
	//Firebird_WriteAlarms(ParamTimeBetweenReconnect:= T#1M);
END_IF

METHOD M_AlarmManager : BOOL
VAR_INPUT
END_VAR

VAR
	KK : UINT;
	
END_VAR
		
		
		
		
// initialisation des AlarmCode et des RecupWord		
	AX_RecupWord[ 1] := A1_PP.MesData.MesAlarmCode; 	
	AX_RecupWord[ 2] := A1_PP.MesData.MesWarningCode; 	
	AX_RecupWord[ 3] := A1_PP.MesData.MesWarningCode2; 	
	AX_RecupWord[ 4] := A1_PP.MesData.MesEventCode;
END_METHOD

METHOD M_AlarmProcessing : BOOL
////////////////// 
// Process alarms, detect changes and segregate if the alarm has to be logged in csv, send by mail, or send by sms
//////////////////


VAR
	LL : UINT;
	KK : UINT;
	
	MesXorWord 		: WORD;
	MesAlarmWord	: WORD;


	IN_AlarmInflux : ST_InfluxAlarmsInsert;
	MesRolAlarmWord: WORD;
	MesRolXoRWord: WORD;
END_VAR
//Retrieve all Alarms word and detect if a change occured. 
FOR KK := 1 TO CstNbAlarmCode DO
	MesXorWord := AX_MesAlarmCode[KK] XOR AX_RecupWord[KK];
	IF MesXorWord > 0 THEN  // Compare si il y a eu des changements dans les alarmes word
		FOR LL := 0 TO 15 DO 
			MesRolXoRWord 	:= ROR(MesXorWord, LL);
			MesRolAlarmWord := ROR(AX_RecupWord[KK], LL);
			
			IF MesRolXoRWord.0 THEN  // Si il y a eu un changement sur le bit
				AX_Journal[KK][LL].Value := MesRolAlarmWord.0; // 
				AX_Journal[KK][LL].TimeStamp_Act:= SYSTEMTIME_TO_STRING(CalLocalTimeStruct);	// On ecrit l'heure du changement
	
				IF (AX_Journal[KK][LL].Value AND AX_Journal[KK][LL].Groupe > 0) OR ( NOT(AX_Journal[KK][LL].Value) AND  AX_Journal[KK][LL].Groupe = 2)  THEN// Il s'agit d'une alarme qu'on doit écrire sur activation

					// CSV alarms :  on ecrit l'alarme
					FUN_Alarms_CSV.FIFO.In := AX_Journal[KK][LL];
					FUN_Alarms_CSV.FIFO.A_Add();
					
					//MAIl alarms
					IF AX_Journal[KK][LL].Alarms_LVL.3 THEN
						FUN_SendMail.FIFO.In := AX_Journal[KK][LL];
						FUN_SendMail.FIFO.A_Add();
					END_IF
					
					InfluxDb_AlarmsManagement.IN_FIFO.In :=  AX_Journal[KK][LL];
					InfluxDb_AlarmsManagement.IN_FIFO.A_Add();
					
					// SMS Alarms. On ecrit si Serveur SMS n'est pas descativé
					IF NOT ParamDisableSMS  AND AX_Journal[KK][LL].Alarms_LVL.4 THEN 
						SMS_Server.IN_DataSetFifo_SendSMS.In.IndexWord		:= KK;
						SMS_Server.IN_DataSetFifo_SendSMS.IN.IndexBit		:= LL;
						SMS_Server.IN_DataSetFifo_SendSMS.IN.Num_tel 		:= '';
						SMS_Server.IN_DataSetFifo_SendSMS.In.ID				:= AX_Journal[KK][LL].ID;
						SMS_Server.IN_DataSetFifo_SendSMS.In.TimeStamp_Act	:= AX_Journal[KK][LL].TimeStamp_Act;						
						SMS_Server.IN_DataSetFifo_SendSMS.IN.Active			:= AX_Journal[KK][LL].Value;	// TRUE si activation. 
						SMS_Server.IN_DataSetFifo_SendSMS.IN.Alarms_LVL		:= AX_Journal[KK][LL].Alarms_LVL ;
						SMS_Server.IN_DataSetFifo_SendSMS.A_Add();
					END_IF 
				END_IF
			END_IF
		END_FOR
		memcpy(destAddr := ADR(AX_MesAlarmCode[KK]), srcAddr :=ADR(AX_RecupWord[KK]), n := SIZEOF(AX_RecupWord[KK])); //On écrase la valeur par la dernière valeur.	
	END_IF
END_FOR
END_METHOD

METHOD M_ForceAlarms : BOOL
VAR_INPUT
END_VAR
// Compteur pour séquencer l'activation des alarmes 		
		
TON_TriggerCount(IN := bTriggerCount, PT := ParamDelayForceAlarm);		
		
F_TRIG_TriggerCount(CLK := bTriggerCount);		
		
IF nCountSequence <= CstNbAlarmCode+1 THEN		
	IF F_TRIG_TriggerCount.Q = TRUE THEN	
		bTriggerCount := TRUE;
	END_IF	
END_IF		
		
IF TON_TriggerCount.Q THEN
	IF nCountSequence < CstNbAlarmCode +1 THEN 
		MesAlarmWordTestJulienDecouple[nCountSequence] := 65535;
	END_IF
	IF nCountSequence-1 > 0 THEN 	
		MesAlarmWordTestJulienDecouple[nCountSequence-1] := 0;
	END_IF	
	nCountSequence := nCountSequence + 1;	
	bTriggerCount := FALSE;	
END_IF		


A1_PP.MesData.MesAlarmCode:= MesAlarmWordTestJulienDecouple[1];
A1_PP.MesData.MesWarningCode:= MesAlarmWordTestJulienDecouple[2];
A1_PP.MesData.MesWarningCode2:= MesAlarmWordTestJulienDecouple[3];
A1_PP.MesData.MesEventCode:= MesAlarmWordTestJulienDecouple[4];
END_METHOD

METHOD M_G7_SMS : BOOL
VAR_IN_OUT
	DataSetFifo_ReadSMS		: FB_SMSDatasetFifo_Read;	
    IN_DataSetFifo_SendSMS		: FB_SMSDatasetFifo_Send;
	CPT_Message				: CTU;
	InStruct 				: ST_ValuesAlarms;
	G7_Etape 				: SINT;
	AX_Numtel				: ARRAY[1..CstNbUser] OF STRING(26);	//Contient tous les numéros des utilisateurs
	AX_Subscribed			: ARRAY[1..CstNbUser] OF BOOL;			//Contient tous les états d'abonnements des utilisateurs aux SMS
	AX_MesAlarmCode_Bool	: ARRAY [1..CstNbAlarmCode] OF ARRAY[1..15] OF BOOL; //Tableau de tous les alarmesCode en Bool
	AX_Cmd_SMS				: ARRAY[1..CstNbCMD] OF STRING(26);
END_VAR

VAR
	Message : STRING(255);
	SUB_MVcalstate			: BYTE;
	SUB_MVData				: SUBMV;
	KK					: INT;
	MM					: INT;
	LL					: INT;
	JJ					: INT;
	ii					: SINT;
	Id_Num				: INT;
	sState				: STRING;

	Etat    			: STRING(255);
	EtatDp1				: STRING(255);
	EtatMainMVCB				: STRING(255);
	FbFormat			: FB_FormatString;
	RestartGsm			: BOOL;
	
	bLocal				: STRING(255);
END_VAR
CPT_Message(PV:=16,CU:=TRUE,RESET:=CPT_Message.Q);
CPT_Message(CU:=FALSE,RESET:=CPT_Message.Q);
CASE G7_Etape OF
	
	1://Commande INFO

		//IF A1_SUBMV.MesDataExd.MesData.MesState.2 THEN 
		//	Etat := 'Decouple, ';
		//ELSIF A1_SUBMV.MesDataExd.MesData.MesState.1 THEN
		//	Etat := 'Couplee, ';
		//ELSIF A1_SUBMV.MesDataExd.MesData.MesState.0 THEN
		//	Etat := 'Effacee, ';
		//END_IF
        //
		//fbFormat(
		//	sFormat:= 'LHERM: %s ; P:%.1f kW; P_PT1: %.1f kW; P_PT2: %.1f kW; P_PT3: %.1f kW; P_PT4: %.1f kW ',
		//	arg1:= F_STRING(Etat), 
		//	arg2:= F_REAL(A1_PP.MesData.MesPsol),  
		//	arg3:= F_REAL(AX_PTR[1].MesDataExd.MesData.MesP), 
		//	arg4:= F_REAL(AX_PTR[2].MesDataExd.MesData.MesP),
		//	arg5:= F_REAL(AX_PTR[3].MesDataExd.MesData.MesP), 
		//	arg6:= F_REAL(AX_PTR[4].MesDataExd.MesData.MesP),
		//	sOut=> Message);
	    //
		//FUN_Alarms.AX_Journal[0][CPT_Message.CV].Message := Message;	
		//IN_DataSetFifo_SendSMS.In.Num_tel:=DataSetFifo_ReadSMS.Out.Num;
		//IN_DataSetFifo_SendSMS.In.IndexWord:=0;
		//IN_DataSetFifo_SendSMS.In.IndexBit:=WORD_TO_SINT(CPT_Message.CV);
		//IN_DataSetFifo_SendSMS.A_Add();
		////DataSetFifo_ReadSMS.A_Remove();
		////2eme message
		//
		//CPT_Message(CU:=TRUE,RESET:=CPT_Message.Q);
		//CPT_Message(CU:=FALSE,RESET:=CPT_Message.Q);
		//fbFormat(
		//	sFormat:= 'Irradiation :PT1GHI: %.1f W/m2; PT1GTI1: %.1f W/m2; PT4GTI_1: %.1f W/m2; PT4GTI_2: %.1f W/m2 ',
		//	arg1:= F_REAl(A1_WS.AX_Pyrano[1].MesData.Value), 
		//	arg2:= F_REAl(A1_WS.AX_Pyrano[2].MesData.Value),   
		//	arg3:= F_REAl(A1_WS.AX_Pyrano[3].MesData.Value), 
		//	arg4:= F_REAl(A1_WS.AX_Pyrano[4].MesData.Value), 
		//	sOut=> Message);
		//	
		//FUN_Alarms.AX_Journal[0][CPT_Message.CV].Message := Message;	
		//IN_DataSetFifo_SendSMS.In.Num_tel:=DataSetFifo_ReadSMS.Out.Num;
		//IN_DataSetFifo_SendSMS.In.IndexWord:=0;
		//IN_DataSetFifo_SendSMS.In.IndexBit:=WORD_TO_SINT(CPT_Message.CV);
		//IN_DataSetFifo_SendSMS.A_Add();
		//
		//////3eme message
		//
		//CPT_Message(CU:=TRUE,RESET:=CPT_Message.Q);
		//CPT_Message(CU:=FALSE,RESET:=CPT_Message.Q);
		//
		//AX_HV_Cel_PDL[1]:= SEL(A1_SUBMV.A1_MainMVCB.MesDataExd.MesData.MesClosed,'Ouvert','Ferme');
		//AX_HV_Cel_PDL[2]:= SEL(A1_SUBMV.AX_FeederMVCB[1].MesDataExd.MesData.MesClosed,'Ouvert','Ferme');
		//AX_HV_Cel_PDL[3]:= SEL(A1_SUBMV.AX_FeederMVCB[1].MesDataExd.MesData.MesClosed,'Ouvert','Ferme');
		//Ax_ETAT_DM1[1]	:= SEL(AX_PTR[1].A1_MainMVCB_PTR.MesDAtaExd.MesData.MesClosed,'Ouvert','Ferme');
		//Ax_ETAT_DM1[2]	:= SEL(AX_PTR[2].A1_MainMVCB_PTR.MesDAtaExd.MesData.MesClosed,'Ouvert','Ferme');
		//Ax_ETAT_DM1[3]	:= SEL(AX_PTR[3].A1_MainMVCB_PTR.MesDAtaExd.MesData.MesClosed,'Ouvert','Ferme');
		//Ax_ETAT_DM1[4]	:= SEL(AX_PTR[4].A1_MainMVCB_PTR.MesDAtaExd.MesData.MesClosed,'Ouvert','Ferme');
		//
		//fbFormat(
		//	sFormat:= 'MainMVCB: %s;  FeederMVCB_1: %s ; FeederMVCB_2: %s; MainMVCB_PTR1: %s;  MainMVCB_PTR2: %s;  MainMVCB_PTR3: %s;  MainMVCB_PTR4: %s  ',
		//	arg1:= F_STRING(AX_HV_Cel_PDL[1]), 
		//	arg2:= F_STRING(AX_HV_Cel_PDL[2]),  
		//	arg3:= F_STRING(AX_HV_Cel_PDL[3]), 
		//	arg4:= F_STRING(Ax_ETAT_DM1[1]), 
		//	arg5:= F_STRING(Ax_ETAT_DM1[2]), 
		//	arg6:= F_STRING(Ax_ETAT_DM1[3]), 
		//	arg7:= F_STRING(Ax_ETAT_DM1[4]), 
		//	sOut=> Message);
	    //
		//FUN_Alarms.AX_Journal[0][CPT_Message.CV].Message := Message;
	    //
		//IN_DataSetFifo_SendSMS.In.Num_tel:=DataSetFifo_ReadSMS.Out.Num;
		//IN_DataSetFifo_SendSMS.In.IndexWord:=0;
		//IN_DataSetFifo_SendSMS.In.IndexBit:=WORD_TO_SINT(CPT_Message.CV);
		//IN_DataSetFifo_SendSMS.A_Add();
		//
		//DataSetFifo_ReadSMS.A_Remove();
		//		
		//InStruct.ID := 975;
		//InStruct.Message :=concat(concat('Le numero de telephone ', IN_DataSetFifo_SendSMS.In.Num_tel), 'a fait une demande Infos par SMS') ;
		//InStruct.TimeStamp_Act := SYSTEMTIME_TO_STRING(CalLocalTimeStruct);
		////FUN_Alarms_CSV.M_AddAction_FIFO(InStruct := InStruct); // Alarme sur activation du code
		//FUN_Alarms_CSV.FIFO.In := InStruct ;
		//FUN_Alarms_CSV.FIFO.A_Add() ;
		
	2://Restart Routeur ADSL
		RestartGsm							:= TRUE;
		OpcUa.AllDataWPulse.CmdReset_Router_ADSL		:= TRUE;
		Message :='Le Routeur Adsl va redemarer';
		FUN_Alarms.AX_Journal[0][CPT_Message.CV].Message := Message;	
		IN_DataSetFifo_SendSMS.In.Num_tel:=DataSetFifo_ReadSMS.Out.Num;
		IN_DataSetFifo_SendSMS.In.IndexWord:=0;
		IN_DataSetFifo_SendSMS.In.IndexBit:=WORD_TO_SINT(CPT_Message.CV);
		IN_DataSetFifo_SendSMS.A_Add();
		DataSetFifo_ReadSMS.A_Remove();
	
		InStruct.ID := 976;
		InStruct.Message := concat(concat('Le numero de telephone ', IN_DataSetFifo_SendSMS.In.Num_tel), 'a Restart le routeur ADSL') ;
		InStruct.TimeStamp_Act := SYSTEMTIME_TO_STRING(CalLocalTimeStruct);
		//FUN_Alarms_CSV.M_AddAction_FIFO(InStruct := InStruct); // Alarme sur activation du code
		FUN_Alarms_CSV.FIFO.In := InStruct ;
		FUN_Alarms_CSV.FIFO.A_Add() ;
		
	3://Puissance des onduleurs
		// 1er message 
		fbFormat(
		sFormat:= 'Onduleur PT1O1: %.1f, PT1O2: %.1f, PT2O1: %.1f, PT2O2: %.1f, PT3O1: %.1f, PT3O2: %.1f, PT4O1: %.1f, PT4O2: %.1f',
		arg1:= F_REAL(Ax_PTR[1].AX_INV[1].MesDataExd.MesData.MesP),
		arg2:= F_REAL(Ax_PTR[1].AX_INV[2].MesDataExd.MesData.MesP),
		arg3:= F_REAL(Ax_PTR[2].AX_INV[1].MesDataExd.MesData.MesP),
		arg4:= F_REAL(Ax_PTR[2].AX_INV[2].MesDataExd.MesData.MesP),
		arg5:= F_REAL(Ax_PTR[3].AX_INV[1].MesDataExd.MesData.MesP),
		arg6:= F_REAL(Ax_PTR[3].AX_INV[2].MesDataExd.MesData.MesP),
		arg7:= F_REAL(Ax_PTR[4].AX_INV[1].MesDataExd.MesData.MesP),
		arg8:= F_REAL(Ax_PTR[4].AX_INV[2].MesDataExd.MesData.MesP),
		sOut=> Message);
		
		FUN_Alarms.AX_Journal[0][CPT_Message.CV].Message := Message;	
		IN_DataSetFifo_SendSMS.In.Num_tel:=DataSetFifo_ReadSMS.Out.Num;
		IN_DataSetFifo_SendSMS.In.IndexWord:=0;
		IN_DataSetFifo_SendSMS.In.IndexBit:= WORD_TO_SINT(CPT_Message.CV);
		IN_DataSetFifo_SendSMS.A_Add();		

		DataSetFifo_ReadSMS.A_Remove();
		
		InStruct.ID := 977;
		InStruct.Message := concat(concat('Le numero de telephone ', IN_DataSetFifo_SendSMS.In.Num_tel), 'a demandé la puissance des onduleurs'); 
		InStruct.TimeStamp_Act := SYSTEMTIME_TO_STRING(CalLocalTimeStruct);
		//FUN_Alarms_CSV.M_AddAction_FIFO(InStruct := InStruct); // Alarme sur activation du code
		FUN_Alarms_CSV.FIFO.In := InStruct ;
		FUN_Alarms_CSV.FIFO.A_Add() ;
		
	4://Mise en pause des alarmes
		ParamDisableSMS := TRUE;
		Message :='Les alarmes SMS sont desactivees';
		FOR MM := 1 TO CstNbUser DO	
			IF AX_Numtel[MM]<>'' THEN
				FUN_Alarms.AX_Journal[0][CPT_Message.CV].Message := Message;	
				IN_DataSetFifo_SendSMS.In.Num_tel:=AX_Numtel[MM];
				IN_DataSetFifo_SendSMS.In.IndexWord:=0;
				IN_DataSetFifo_SendSMS.In.IndexBit:= WORD_TO_SINT(CPT_Message.CV);
				IN_DataSetFifo_SendSMS.A_Add();
				DataSetFifo_ReadSMS.A_Remove();
			END_IF
		END_FOR
		
		InStruct.ID := 978;
		InStruct.Message := concat(concat('Le numero de telephone ', IN_DataSetFifo_SendSMS.In.Num_tel), 'a désactivé les alarmes SMS'); 
		InStruct.TimeStamp_Act := SYSTEMTIME_TO_STRING(CalLocalTimeStruct);
		//FUN_Alarms_CSV.M_AddAction_FIFO(InStruct := InStruct); // Alarme sur activation du code
		FUN_Alarms_CSV.FIFO.In := InStruct ;
		FUN_Alarms_CSV.FIFO.A_Add() ;
	
	5://Start SMS
		ParamDisableSMS := FALSE;
		Message :='Les alarmes SMS sont activees';
		FOR MM := 1 TO CstNbUser DO	
			IF AX_Numtel[MM]<>'' THEN
				FUN_Alarms.AX_Journal[0][CPT_Message.CV].Message := Message;	
				IN_DataSetFifo_SendSMS.In.Num_tel:=AX_Numtel[MM];
				IN_DataSetFifo_SendSMS.In.IndexWord:=0;
				IN_DataSetFifo_SendSMS.In.IndexBit:= WORD_TO_SINT(CPT_Message.CV);
				IN_DataSetFifo_SendSMS.A_Add();
				DataSetFifo_ReadSMS.A_Remove();
			END_IF
		END_FOR
		
		InStruct.ID := 979;
		InStruct.Message := concat(concat('Le numero de telephone ', IN_DataSetFifo_SendSMS.In.Num_tel), 'a réactivé les alarmes SMS'); 
		InStruct.TimeStamp_Act := SYSTEMTIME_TO_STRING(CalLocalTimeStruct);
		//FUN_Alarms_CSV.M_AddAction_FIFO(InStruct := InStruct); // Alarme sur activation du code
		FUN_Alarms_CSV.FIFO.In := InStruct ;
		FUN_Alarms_CSV.FIFO.A_Add() ;
	

 	6:// Unsubscribe
		FOR LL := 1 TO CstNbUser DO
			IF DataSetFifo_ReadSMS.Out.Num = AX_Numtel[LL] THEN
				Id_Num := LL;
				EXIT;
			END_IF
		END_FOR
		AX_Subscribed[Id_Num] := NOT AX_Subscribed[Id_Num];
		sState := SEL(AX_Subscribed[Id_Num], 'Unsubscribed', 'Subscribed');
		Message := Concat('You have toggled your subscription, state =', sState);
		FUN_Alarms.AX_Journal[0][CPT_Message.CV].Message := Message ;
		IN_DataSetFifo_SendSMS.In.Num_tel:=DataSetFifo_ReadSMS.Out.Num;
		IN_DataSetFifo_SendSMS.In.IndexWord:=0;
		IN_DataSetFifo_SendSMS.In.IndexBit:= WORD_TO_SINT(CPT_Message.CV);
		IN_DataSetFifo_SendSMS.A_Add();
		DataSetFifo_ReadSMS.A_Remove();
		
		InStruct.ID := 980;
		InStruct.Message := concat(concat('Le numero de telephone ', IN_DataSetFifo_SendSMS.In.Num_tel), 'a modifie son inscription') ;
		InStruct.TimeStamp_Act := SYSTEMTIME_TO_STRING(CalLocalTimeStruct);
		//FUN_Alarms_CSV.M_AddAction_FIFO(InStruct := InStruct); // Alarme sur activation du code
		FUN_Alarms_CSV.FIFO.In := InStruct ;
		FUN_Alarms_CSV.FIFO.A_Add() ;
		
	7 : 	//Get Public IP 
		fbFormat(
			sFormat:= 'IP publique de la centrale : %s',
			arg1:= F_STRING(ParamIpPublic),
			sOut=> Message);
		
		FUN_Alarms.AX_Journal[0][CPT_Message.CV].Message := Message;	
		IN_DataSetFifo_SendSMS.In.Num_tel:=DataSetFifo_ReadSMS.Out.Num;
		IN_DataSetFifo_SendSMS.In.IndexWord:=0;
		IN_DataSetFifo_SendSMS.In.IndexBit:= WORD_TO_SINT(CPT_Message.CV);
		IN_DataSetFifo_SendSMS.A_Add();
		DataSetFifo_ReadSMS.A_Remove();
		CPT_Message(CU:=TRUE,RESET:=CPT_Message.Q);
		CPT_Message(CU:=FALSE,RESET:=CPT_Message.Q);
		
		InStruct.ID := 981;
		InStruct.Message := concat(concat('Le numero de telephone ', IN_DataSetFifo_SendSMS.In.Num_tel), 'a demandé l IP public ');  
		InStruct.TimeStamp_Act := SYSTEMTIME_TO_STRING(CalLocalTimeStruct);
		//FUN_Alarms_CSV.M_AddAction_FIFO(InStruct := InStruct); // Alarme sur activation du code
		FUN_Alarms_CSV.FIFO.In := InStruct ;
		FUN_Alarms_CSV.FIFO.A_Add() ; 
		
	8: // All Active Alarms
		FOR jj := 1 TO CstNbAlarmCode DO
			FOR ii :=1 TO 15 DO 
				IF(AX_Journal[jj][ii].Value AND (AX_Journal[jj][ii].Alarms_LVL.0 OR AX_Journal[jj][ii].Alarms_LVL.1) AND AX_Journal[jj][ii].Groupe > 0 AND NOT ParamDisableSMS ) THEN // Il s'agit d'une alarme qu'on doit notifier par sms
					IN_DataSetFifo_SendSMS.In.IndexWord	:= jj;
					IN_DataSetFifo_SendSMS.IN.IndexBit		:= ii;
					IN_DataSetFifo_SendSMS.In.Num_tel		:= DataSetFifo_ReadSMS.Out.Num;
					IN_DataSetFifo_SendSMS.IN.Active		:= TRUE;
					IN_DataSetFifo_SendSMS.A_Add();
					CPT_Message(CU:=TRUE,RESET:=CPT_Message.Q);
					CPT_Message(CU:=FALSE,RESET:=CPT_Message.Q);
				END_IF
			END_FOR
		END_FOR
		DataSetFifo_ReadSMS.A_Remove();
		
		InStruct.ID := 982;
		InStruct.Message := concat(concat('Le numero de telephone ', IN_DataSetFifo_SendSMS.In.Num_tel), 'a demandé la liste des alarmes actives');  
		InStruct.TimeStamp_Act := SYSTEMTIME_TO_STRING(CalLocalTimeStruct);
		//FUN_Alarms_CSV.M_AddAction_FIFO(InStruct := InStruct); // Alarme sur activation du code
		FUN_Alarms_CSV.FIFO.In := InStruct ;
		FUN_Alarms_CSV.FIFO.A_Add() ;
		
	9: // Help
		Message :='Les commandes disponibles sont :Infos ';
		FOR KK := 2 TO MIN(7,CstNbCMD) DO // Nbr_CMD-1 DO //pas besoin du Help
			Message := concat(Message, concat('", "',  AX_Cmd_SMS[KK]));
		END_FOR
		FUN_Alarms.AX_Journal[0][CPT_Message.CV].Message := Message;	
		IN_DataSetFifo_SendSMS.In.Num_tel:=DataSetFifo_ReadSMS.Out.Num;
		IN_DataSetFifo_SendSMS.In.IndexWord:=0;
		IN_DataSetFifo_SendSMS.In.IndexBit:=WORD_TO_SINT(CPT_Message.CV);
		IN_DataSetFifo_SendSMS.A_Add();
		
		IF CstNbCMD >7 THEN
			CPT_Message(CU:=TRUE,RESET:=CPT_Message.Q);
			CPT_Message(CU:=FALSE,RESET:=CPT_Message.Q);

			Message :='';
			FOR KK := 8 TO MIN(14,CstNbCMD) DO // Nbr_CMD-1 DO //pas besoin du Help
				Message := concat(Message, concat('", "',  AX_Cmd_SMS[KK]));
			END_FOR	
			FUN_Alarms.AX_Journal[0][CPT_Message.CV].Message := Message;	
			IN_DataSetFifo_SendSMS.In.Num_tel:=DataSetFifo_ReadSMS.Out.Num;
			IN_DataSetFifo_SendSMS.In.IndexWord:=0;
			IN_DataSetFifo_SendSMS.In.IndexBit:=WORD_TO_SINT(CPT_Message.CV);
			IN_DataSetFifo_SendSMS.A_Add();				
		END_IF
		
		IF CstNbCMD >14 THEN
			CPT_Message(CU:=TRUE,RESET:=CPT_Message.Q);
			CPT_Message(CU:=FALSE,RESET:=CPT_Message.Q);

			Message :='';
			FOR KK := 14 TO CstNbCMD DO // Nbr_CMD-1 DO //pas besoin du Help
				Message := concat(Message, concat('", "',  AX_Cmd_SMS[KK]));
			END_FOR	
			FUN_Alarms.AX_Journal[0][CPT_Message.CV].Message := Message;	
			IN_DataSetFifo_SendSMS.In.Num_tel:=DataSetFifo_ReadSMS.Out.Num;
			IN_DataSetFifo_SendSMS.In.IndexWord:=0;
			IN_DataSetFifo_SendSMS.In.IndexBit:=WORD_TO_SINT(CPT_Message.CV);
			IN_DataSetFifo_SendSMS.A_Add();				
		END_IF
		
		DataSetFifo_ReadSMS.A_Remove();
			
		InStruct.ID := 983;
		InStruct.Message := concat(concat('Le numero de telephone ', IN_DataSetFifo_SendSMS.In.Num_tel), 'a demandé la commande Help'); 
		InStruct.TimeStamp_Act := SYSTEMTIME_TO_STRING(CalLocalTimeStruct);
		//FUN_Alarms_CSV.M_AddAction_FIFO(InStruct := InStruct); // Alarme sur activation du code
		FUN_Alarms_CSV.FIFO.In := InStruct ;
		FUN_Alarms_CSV.FIFO.A_Add() ;
	
10: // test d'envois sms
		OPCUA.AllDataWPulse.CmdTestSms := TRUE;
		DataSetFifo_ReadSMS.A_Remove();
		
		InStruct.ID := 984;
		InStruct.Message := concat(concat('Le numero de telephone ', IN_DataSetFifo_SendSMS.In.Num_tel), 'a envoyé une cmd test sms et mail'); 
		InStruct.TimeStamp_Act := SYSTEMTIME_TO_STRING(CalLocalTimeStruct);
		//FUN_Alarms_CSV.M_AddAction_FIFO(InStruct := InStruct); // Alarme sur activation du code
		FUN_Alarms_CSV.FIFO.In := InStruct ;
		FUN_Alarms_CSV.FIFO.A_Add() ;
		
	11: //Forced stay connect Toggle
		A1_PP.ParamForcedStayConnect := NOT A1_PP.ParamForcedStayConnect;
		sState := SEL(A1_PP.ParamForcedStayConnect, 'False', 'True');
		Message := Concat('You have toggled the Variable ForcedStayConnect, state =', sState);
		FUN_Alarms.AX_Journal[0][CPT_Message.CV].Message := Message ;
		IN_DataSetFifo_SendSMS.In.Num_tel:=DataSetFifo_ReadSMS.Out.Num;
		IN_DataSetFifo_SendSMS.In.IndexWord:=0;
		IN_DataSetFifo_SendSMS.In.IndexBit:= WORD_TO_SINT(CPT_Message.CV);
		IN_DataSetFifo_SendSMS.A_Add();
		DataSetFifo_ReadSMS.A_Remove();
		
		InStruct.ID := 985;
		InStruct.Message := concat(concat('Le numero de telephone ', IN_DataSetFifo_SendSMS.In.Num_tel), 'a modifie la variable ForceStauConnect') ;
		InStruct.TimeStamp_Act := SYSTEMTIME_TO_STRING(CalLocalTimeStruct);
		//FUN_Alarms_CSV.M_AddAction_FIFO(InStruct := InStruct); // Alarme sur activation du code
		FUN_Alarms_CSV.FIFO.In := InStruct ;
		FUN_Alarms_CSV.FIFO.A_Add() ;
	
	12: // Restart HH
		OPCUA.AllDataWPulse.CmdRestart_Telegraf := TRUE;
		Message := 'Telegraf is restarting';
		FUN_Alarms.AX_Journal[0][CPT_Message.CV].Message := Message ;
		IN_DataSetFifo_SendSMS.In.Num_tel:=DataSetFifo_ReadSMS.Out.Num;
		IN_DataSetFifo_SendSMS.In.IndexWord:=0;
		IN_DataSetFifo_SendSMS.In.IndexBit:= WORD_TO_SINT(CPT_Message.CV);
		IN_DataSetFifo_SendSMS.A_Add();
		DataSetFifo_ReadSMS.A_Remove();
		
		InStruct.ID := 986;
		InStruct.Message := concat(concat('Le numero de telephone ', IN_DataSetFifo_SendSMS.In.Num_tel), 'a redemarre le service Telegraf') ;
		InStruct.TimeStamp_Act := SYSTEMTIME_TO_STRING(CalLocalTimeStruct);
		//FUN_Alarms_CSV.M_AddAction_FIFO(InStruct := InStruct); // Alarme sur activation du code
		FUN_Alarms_CSV.FIFO.In := InStruct ;
		FUN_Alarms_CSV.FIFO.A_Add() ;
	
	13: // Restart PLC
		OPCUA.AllDataWPulse.CmdRestart_PLC := TRUE;
		Message := 'PLC is restarting Now !';
		FUN_Alarms.AX_Journal[0][CPT_Message.CV].Message := Message ;
		IN_DataSetFifo_SendSMS.In.Num_tel:=DataSetFifo_ReadSMS.Out.Num;
		IN_DataSetFifo_SendSMS.In.IndexWord:=0;
		IN_DataSetFifo_SendSMS.In.IndexBit:= WORD_TO_SINT(CPT_Message.CV);
		IN_DataSetFifo_SendSMS.A_Add();
		DataSetFifo_ReadSMS.A_Remove();
		
		InStruct.ID := 987;
		InStruct.Message := concat(concat('Le numero de telephone ', IN_DataSetFifo_SendSMS.In.Num_tel), 'a redemarre le PLC') ;
		InStruct.TimeStamp_Act := SYSTEMTIME_TO_STRING(CalLocalTimeStruct);
		//FUN_Alarms_CSV.M_AddAction_FIFO(InStruct := InStruct); // Alarme sur activation du code
		FUN_Alarms_CSV.FIFO.In := InStruct ;
		FUN_Alarms_CSV.FIFO.A_Add() ;
		
	14: // autorisation de couplage
		OpcUa.AllDataWPulse.CmdAutCpl := TRUE;
		
		Message := 'Autorisation de couplage recu';
		FUN_Alarms.AX_Journal[0][CPT_Message.CV].Message := Message ;
		IN_DataSetFifo_SendSMS.In.Num_tel:=DataSetFifo_ReadSMS.Out.Num;
		IN_DataSetFifo_SendSMS.In.IndexWord:=0;
		IN_DataSetFifo_SendSMS.In.IndexBit:= WORD_TO_SINT(CPT_Message.CV);
		IN_DataSetFifo_SendSMS.A_Add();
		DataSetFifo_ReadSMS.A_Remove();
		
		InStruct.ID := 988;
		InStruct.Message := concat(concat('Le numero de telephone ', IN_DataSetFifo_SendSMS.In.Num_tel), 'a envoye une autorisation de couplage') ;
		InStruct.TimeStamp_Act := SYSTEMTIME_TO_STRING(CalLocalTimeStruct);
		//FUN_Alarms_CSV.M_AddAction_FIFO(InStruct := InStruct); // Alarme sur activation du code
		FUN_Alarms_CSV.FIFO.In := InStruct ;
		FUN_Alarms_CSV.FIFO.A_Add() ;
		
	15: // Disconnect order
		OPCUA.AllDataWPulse.CmdDisconnect  := TRUE;
		Message := 'Ordre de decouplage recu';
		FUN_Alarms.AX_Journal[0][CPT_Message.CV].Message := Message ;
		IN_DataSetFifo_SendSMS.In.Num_tel:=DataSetFifo_ReadSMS.Out.Num;
		IN_DataSetFifo_SendSMS.In.IndexWord:=0;
		IN_DataSetFifo_SendSMS.In.IndexBit:= WORD_TO_SINT(CPT_Message.CV);
		IN_DataSetFifo_SendSMS.A_Add();
		DataSetFifo_ReadSMS.A_Remove();
		
		InStruct.ID := 989;
		InStruct.Message := concat(concat('Le numero de telephone ', IN_DataSetFifo_SendSMS.In.Num_tel), ' a fait une demande de decouplage') ;
		InStruct.TimeStamp_Act := SYSTEMTIME_TO_STRING(CalLocalTimeStruct);
		//InStruct
		//FUN_Alarms_CSV.M_AddAction_FIFO(InStruct := InStruct); // Alarme sur activation du code
		FUN_Alarms_CSV.FIFO.In := InStruct ;
		FUN_Alarms_CSV.FIFO.A_Add() ;
	16: // Connect VPN
		OpcUa.AllDataWPulse.CmdStart_Vpn := TRUE;
		Message := 'Starting VPN';
		FUN_Alarms.AX_Journal[0][CPT_Message.CV].Message := Message ;
		IN_DataSetFifo_SendSMS.In.Num_tel:=DataSetFifo_ReadSMS.Out.Num;
		IN_DataSetFifo_SendSMS.In.IndexWord:=0;
		IN_DataSetFifo_SendSMS.In.IndexBit:= WORD_TO_SINT(CPT_Message.CV);
		IN_DataSetFifo_SendSMS.A_Add();
		DataSetFifo_ReadSMS.A_Remove();
		
		InStruct.ID := 990;
		InStruct.Message := concat(concat('Le numero de telephone ', IN_DataSetFifo_SendSMS.In.Num_tel), ' a lance le VPN') ;
		InStruct.TimeStamp_Act := SYSTEMTIME_TO_STRING(CalLocalTimeStruct);
		//InStruct
		//FUN_Alarms_CSV.M_AddAction_FIFO(InStruct := InStruct); // Alarme sur activation du code
		FUN_Alarms_CSV.FIFO.In := InStruct ;
		FUN_Alarms_CSV.FIFO.A_Add() ;
	
	17: // Disconnect VPN
		OpcUa.AllDataWPulse.CmdStop_Vpn := TRUE;
		Message := 'Stopping VPN';
		FUN_Alarms.AX_Journal[0][CPT_Message.CV].Message := Message ;
		IN_DataSetFifo_SendSMS.In.Num_tel:=DataSetFifo_ReadSMS.Out.Num;
		IN_DataSetFifo_SendSMS.In.IndexWord:=0;
		IN_DataSetFifo_SendSMS.In.IndexBit:= WORD_TO_SINT(CPT_Message.CV);
		IN_DataSetFifo_SendSMS.A_Add();
		DataSetFifo_ReadSMS.A_Remove();
		
		InStruct.ID := 991;
		InStruct.Message := concat(concat('Le numero de telephone ', IN_DataSetFifo_SendSMS.In.Num_tel), ' a arrete le VPN') ;
		InStruct.TimeStamp_Act := SYSTEMTIME_TO_STRING(CalLocalTimeStruct);
		//InStruct
		FUN_Alarms_CSV.FIFO.In := InStruct ;
		FUN_Alarms_CSV.FIFO.A_Add() ;
		
	18: // Reboot IPC
		OpcUa.AllDataWPulse.CmdReset_IPC := TRUE;
		Message :='Le PC industriel va redemarer';
		FUN_Alarms.AX_Journal[0][CPT_Message.CV].Message := Message;	
		IN_DataSetFifo_SendSMS.In.Num_tel:=DataSetFifo_ReadSMS.Out.Num;
		IN_DataSetFifo_SendSMS.In.IndexWord:=0;
		IN_DataSetFifo_SendSMS.In.IndexBit:=WORD_TO_SINT(CPT_Message.CV);
		IN_DataSetFifo_SendSMS.A_Add();
		DataSetFifo_ReadSMS.A_Remove();		
END_CASE
END_METHOD

METHOD M_Init : BOOL
VAR_INPUT
END_VAR

VAR

	KK: INT;
	NbrAlarmCodeCSV: INT;
	LL: INT;
	AX_Jou: INT;
END_VAR
// Minit 


FOR KK := 0 TO CstNbAlarmCode DO			
	FOR LL := 0 TO 15 DO		
		AX_Journal[KK][LL].ID := INT_TO_UINT((KK)*16 + LL);	
		AX_Journal[KK][LL].Message := '';	
		AX_Journal[KK][LL].Groupe := 0;	
		AX_Journal[KK][LL].Alarms_LVL := 0;	
	END_FOR		
END_FOR			
			
			
	AX_Journal[ 1][ 1].Message := 'PP : Impossible to disconnect the power plant';	AX_Journal[ 1][1].Groupe := 1;	AX_Journal[ 1][1].Alarms_LVL := 25;
	AX_Journal[ 1][ 2].Message := 'PP : Redundancy is forced on the other PLC        ';	AX_Journal[ 1][2].Groupe := 1;	AX_Journal[ 1][2].Alarms_LVL := 281;
	AX_Journal[ 1][ 3].Message := 'PP : This PLC is forced in RUN ( redundancy inhibited )     ';	AX_Journal[ 1][3].Groupe := 1;	AX_Journal[ 1][3].Alarms_LVL := 281;
	AX_Journal[ 1][ 4].Message := 'PP : IEC 104 LOC is inhibited. It does not trigger change of PLC   ';	AX_Journal[ 1][4].Groupe := 1;	AX_Journal[ 1][4].Alarms_LVL := 281;
	AX_Journal[ 1][ 5].Message := 'PP : Code is in Test Mode ( Writing order by COM and IO inhibited )   ';	AX_Journal[ 1][5].Groupe := 1;	AX_Journal[ 1][5].Alarms_LVL := 281;
	AX_Journal[ 2][ 1].Message := 'PP : Ping Host Error         ';	AX_Journal[ 2][1].Groupe := 1;	AX_Journal[ 2][1].Alarms_LVL := 266;
	AX_Journal[ 2][ 2].Message := 'PP : SMS server is disabled';	AX_Journal[ 2][2].Groupe := 1;	AX_Journal[ 2][2].Alarms_LVL := 10;
	AX_Journal[ 2][ 3].Message := 'PP : SMS server is enabled';	AX_Journal[ 2][3].Groupe := 1;	AX_Journal[ 2][3].Alarms_LVL := 10;
	AX_Journal[ 2][ 5].Message := 'PP : C drive almost full       ';	AX_Journal[ 2][5].Groupe := 1;	AX_Journal[ 2][5].Alarms_LVL := 266;
	AX_Journal[ 2][ 6].Message := 'PP : Max time reached for decoupling request';	AX_Journal[ 2][6].Groupe := 1;	AX_Journal[ 2][6].Alarms_LVL := 10;
	AX_Journal[ 2][ 7].Message := 'PP : Force Stay connect active      ';	AX_Journal[ 2][7].Groupe := 1;	AX_Journal[ 2][7].Alarms_LVL := 266;
	AX_Journal[ 2][ 8].Message := 'PP : License dongle is missing      ';	AX_Journal[ 2][8].Groupe := 1;	AX_Journal[ 2][8].Alarms_LVL := 266;
	AX_Journal[ 2][ 9].Message := 'PP : PLC CPU usage is above 50%      ';	AX_Journal[ 2][9].Groupe := 1;	AX_Journal[ 2][9].Alarms_LVL := 266;
	AX_Journal[ 2][ 10].Message := 'PP : Force Stay connect is deactivated     ';	AX_Journal[ 2][10].Groupe := 1;	AX_Journal[ 2][10].Alarms_LVL := 266;
	AX_Journal[ 2][ 12].Message := 'PP : Test mode is disabled (outputs reactivated)  ';	AX_Journal[ 2][12].Groupe := 1;	AX_Journal[ 2][12].Alarms_LVL := 266;
	AX_Journal[ 2][ 13].Message := 'PP : Child Warning Synthesis';	AX_Journal[ 2][13].Groupe := 1;	AX_Journal[ 2][13].Alarms_LVL := 10;
	AX_Journal[ 2][ 14].Message := 'PP : Test mode enable (outputs inhibited)   ';	AX_Journal[ 2][14].Groupe := 1;	AX_Journal[ 2][14].Alarms_LVL := 266;
	AX_Journal[ 2][ 15].Message := 'PP : Test SMS';	AX_Journal[ 2][15].Groupe := 1;	AX_Journal[ 2][15].Alarms_LVL := 10;
	AX_Journal[ 3][ 1].Message := 'PP : No internet access  ';	AX_Journal[ 3][1].Groupe := 1;	AX_Journal[ 3][1].Alarms_LVL := 33034;
	AX_Journal[ 3][ 2].Message := 'PP : Router not reachable  ';	AX_Journal[ 3][2].Groupe := 1;	AX_Journal[ 3][2].Alarms_LVL := 33034;
	AX_Journal[ 3][ 3].Message := 'PP : SMS Router not reachable  ';	AX_Journal[ 3][3].Groupe := 1;	AX_Journal[ 3][3].Alarms_LVL := 33034;
	AX_Journal[ 3][ 4].Message := 'PP : Industrial PC not reachable  ';	AX_Journal[ 3][4].Groupe := 1;	AX_Journal[ 3][4].Alarms_LVL := 33034;
	AX_Journal[ 3][ 6].Message := 'PP : HMI server not running ';	AX_Journal[ 3][6].Groupe := 1;	AX_Journal[ 3][6].Alarms_LVL := 266;
	AX_Journal[ 3][ 7].Message := 'PP : Open VPN not running  ';	AX_Journal[ 3][7].Groupe := 1;	AX_Journal[ 3][7].Alarms_LVL := 266;
	AX_Journal[ 3][ 8].Message := 'PP : Teamviewer not running ';	AX_Journal[ 3][8].Groupe := 1;	AX_Journal[ 3][8].Alarms_LVL := 266;
	AX_Journal[ 3][ 9].Message := 'PP : OPC UA not running ';	AX_Journal[ 3][9].Groupe := 1;	AX_Journal[ 3][9].Alarms_LVL := 266;
	AX_Journal[ 3][ 10].Message := 'PP : Chronograf not running ';	AX_Journal[ 3][10].Groupe := 1;	AX_Journal[ 3][10].Alarms_LVL := 266;
	AX_Journal[ 3][ 11].Message := 'PP : Telegraf not running ';	AX_Journal[ 3][11].Groupe := 1;	AX_Journal[ 3][11].Alarms_LVL := 266;
	AX_Journal[ 3][ 12].Message := 'PP : InfluxDB not running  ';	AX_Journal[ 3][12].Groupe := 1;	AX_Journal[ 3][12].Alarms_LVL := 266;
	AX_Journal[ 3][ 14].Message := 'PP : Modbus Server not running  ';	AX_Journal[ 3][14].Groupe := 1;	AX_Journal[ 3][14].Alarms_LVL := 266;
	AX_Journal[ 4][ 14].Message := 'PP : Global Init Command';	AX_Journal[ 4][14].Groupe := 1;	AX_Journal[ 4][14].Alarms_LVL := 4;
	AX_Journal[ 4][ 15].Message := 'PP : Global Fault Clear command';	AX_Journal[ 4][15].Groupe := 1;	AX_Journal[ 4][15].Alarms_LVL := 4;
END_METHOD

END_PROGRAM

// ---- 00_FunctionsBlocks/Beckhoff/AlarmManagement/FUN_Alarms_CSV.TcPOU
PROGRAM FUN_Alarms_CSV
////////////////// 
// Save Alarms in a CSV File locally. 
//////////////////	
VAR_INPUT
	ParamSeparateur			: STRING := ';';				// Separator for the CSV file
	ParamExtension			: STRING(255) := '.csv';				// File extension
	FIFO					: FB_DBDatasetFifo;	// Buffer that contains all the alarms to be written in the file. 
		MesData		: ServerCSV ;			//  Server info
END_VAR
VAR_OUTPUT
	
END_VAR
VAR
	format_string				: FB_Formatstring;
	CalDate						: T_MaxString;
	
	// Alarm management 
		bWriteAlarm				: BOOL;				// Writing CSV File failed 
		TON_WritealarmFile		: TON;				// Tempo to detect error in file creation.  
		
		
	// Data processing 

	CalFileName			: STRING;				// Name of csv file 
	
	//Time Values 
	
	//Test existence file 
	FindFile 			: FB_EnumFindFileEntry ;
	FileInfo			: ST_FindFileEntry;
	bFileOK				: BOOL:= TRUE ;

	//Initial File creation 
	GetHostName			: FB_GetHostName;
	WriteFile			: FB_WriteFile;
	bStartWrite			: BOOL;
	bInitWrite			: BOOL;
	
	//Initial File creation 
	InitLine			: T_MaxString;
	LastInitLine		: T_MaxString;
	WelcomeMessage 		: T_MaxString := 'Daily alarms file';
	ForDay				: T_MaxString := 'for day :';
	ForPlant	 		: T_MaxString := 'for plant : ';
	NewLineVar			: T_MaxString := '$L $00';
	TimeStampVar		: T_MaxString := 'TimeStamp;AlarmsID;Description;Activated;Acknowledged;Level;$L$00';
	MessageInitial		: ARRAY[1..10] OF STRING(255);
	MessageInitial_Null	: ARRAY[1..10] OF STRING(255);
	bInitWriting		: BOOL;
	len_to_write		: INT;
	len_to_add			: INT;

	// Write File
	LineToWrite			: STRING(1000);

	// General variables
		bInit 			: BOOL;
		MesTimeStamp 	: STRING(19);				// Timestamp of the alarm
		bOutCompleted 	: RS;						// Writing file is completed
	
	//TABLEAU
		CalTimeStamp: STRING(255);				// Timestamp formatted

END_VAR

IF NOT bInit THEN
	M_Init();
END_IF

M_AlarmManager();

format_string(
	sFormat := 'ALARMS_%0.2d-%0.2d-%0.2d%s', 
	arg1 := F_WORD(in:=CalLocalTimeStruct.wYear),	arg2 := F_WORD(in:=CalLocalTimeStruct.wMonth),	arg3 := F_WORD(in:=CalLocalTimeStruct.wDay),
	arg4 := F_STRING(in:=ParamExtension),
	sOut => CalFileName
);

format_string(
	sFormat := '%0.2d-%0.2d-%0.2d', 
	arg1 := F_WORD(in:=CalLocalTimeStruct.wYear),	arg2 := F_WORD(in:=CalLocalTimeStruct.wMonth),	arg3 := F_WORD(in:=CalLocalTimeStruct.wDay),
	sOut => CalDate
);

InitLine := concat(str1:=WelcomeMessage, STR2:= concat(str1:=
	ParamSeparateur, str2:=concat(STR1:=ForDay, STR2:=concat(str1:= ParamSeparateur, STR2:= concat(str1:= 
	CalDate,str2:=concat(str1:= ParamSeparateur, str2 := CONCAT(str1:=
	ForPlant,str2:=Concat(str1:=ParamSeparateur, str2:= CONCAT(str1:= GetHostName.sHostName, str2:=ParamSeparateur)
))))))));

IF InitLine <> LastInitLine OR InitLine = '' OR (NOT FindFile.bError AND NOT bFileOK) THEN
	LastInitLine := InitLine;
	bInitWriting := TRUE;
END_IF
		
//Test Existence File
IF FUN_CreateDir_CSV.bDirOk THEN
	FindFile
	(
		sNetId := '',
		sPathName := concat(FUN_CreateDir_CSV.AX_DirNames[2],CalFileName),
		eCmd := eEnumCmd_First,
		bExecute := TRUE,
		tTimeout := T#3S,
		stFindFile => FileInfo
	);
	
 MesData.TimeCreation 	:= FILETIME_TO_SYSTEMTIME(filetime := FileInfo.creationTime);
MesData.TimeModif	 	:= FILETIME_TO_SYSTEMTIME(filetime := FileInfo.lastWriteTime);
	
MesData.FileSize  		:= ULARGE_TO_ULINT(in := FileInfo.fileSize);
	IF NOT FindFile.bBusy THEN
		FindFile(bExecute := FALSE);
		bFileOK := MesData.FileSize > 0 ; 
	END_IF
	
	
	IF NOT FindFile.bBusy AND NOT bFileOK AND bInitWriting THEN
		// je réinitialise les longueurs
		len_to_write := 0;
		MessageInitial := MessageInitial_Null;
		MEMCPY(destAddr := ADR(MessageInitial)+len_to_write, srcAddr := ADR(InitLine), n := len(InitLine));
		len_to_add := len(InitLine);			len_to_write := len_to_write + len_to_add;
		
		MEMCPY(destAddr := ADR(MessageInitial)+len_to_write, srcAddr := ADR(NewLineVar), n := len(NewLineVar));
		len_to_add := len(NewLineVar);			len_to_write := len_to_write + len_to_add;
		
		MEMCPY(destAddr := ADR(MessageInitial)+len_to_write, srcAddr := ADR(TimeStampVar), n := len(TimeStampVar));
		len_to_add := len(TimeStampVar);		len_to_write := len_to_write + len_to_add;
		
		WriteFile
		(
			InStart := TRUE,
			InDirFile := concat(FUN_CreateDir_CSV.AX_DirNames[2], CalFileName),
			InAmsId := '', 
			InPMessage := ADR(MessageInitial),
			InLMessage := len_to_write
		);
		
		IF WriteFile.OutCompleted OR bFileOK THEN
			WriteFile(InStart := FALSE);
		END_IF
	END_IF
	
	
	IF bFileOK AND MesData.FileSize < 100000000 AND fifo.nCount > 0 THEN
		bInitWriting := FALSE;
		fifo.A_Get();	// Unpile the buffer to get the next alarm to write. 
		
		MesTimeStamp := CONCAT(REPLACE(STR1:= left(str := FIFO.Out.TimeStamp_Act, 19), STR2 := ' ', L := 1, P := 11), ' ') ;	// Get Timestamp of the activation or desactivation of the alarm
		ReplaceAll( In_StringTosearch := MesTimeStamp, In_StringToFind := '/', IN_StringToReplace := '-', OUT_StringToSearch => CalTimeStamp);
		
		// Create line content
		LineToWrite := Concat(CalTimeStamp, ParamSeparateur);
		LineToWrite := concat(LineToWrite, Concat(STR1 := UINT_TO_STRING(FIFO.Out.ID) ,ParamSeparateur));
		LineToWrite := concat(LineToWrite, Concat(STR1 := FIFO.Out.Message ,ParamSeparateur));
		LineToWrite := Concat(STR1 := LineToWrite, STR2 := Concat(STR1 := BOOL_TO_STRING( FIFO.Out.Value), STR2 := ParamSeparateur));
		LineToWrite:= Concat(STR1 := LineToWrite, Concat(STR1 := BOOL_TO_STRING( FIFO.Out.Ack), STR2 := ParamSeparateur)); 
		LineToWrite:= Concat(STR1 := LineToWrite, Concat(STR1 := UINT_TO_STRING( FIFO.Out.Alarms_LVL), STR2 := ParamSeparateur)); 
		LineToWrite := Concat(LineToWrite, '$L$00');
		
		// Write File
		WriteFile
		(
			InStart := TRUE,
			InDirFile := concat(FUN_CreateDir_CSV.AX_DirNames[2], CalFileName),
			InAmsId := '', 
			InPMessage := ADR(LineToWrite),
			InLMessage := LEN(LineToWrite)
		);
		IF NOT WriteFile.OutBusy AND NOT WriteFile.OutError AND WriteFile.OutCompleted THEN
			// File has been writen successfully
			fifo.A_Remove();
			WriteFile(InStart := FALSE);
			bWriteAlarm	:= FALSE ;
		ELSIF WriteFile.OutError THEN 
			// In case of writing error, try again to write the alarm. 
			bWriteAlarm	:= TRUE ;
			WriteFile(InStart := FALSE);
		END_IF
	END_IF
END_IF

METHOD M_AlarmManager
VAR

	FB_AlarmCodeManager			: FB_AlarmCodeManager ;

END_VAR

TON_WritealarmFile(IN:= NOT bFileOK  , PT:= T#10S  ) ;


// ALARM CODE //
	FB_AlarmCodeManager(
		bAlarm1			:= bWriteAlarm	  ,				// Write CSV Alarm
		bAlarm2			:= fifo.bOverwrite   ,			// Overflow buffer
		bAlarm3			:= TON_WritealarmFile.Q   ,		// Can not create CSV Alarm file 
		bAlarm4			:= FALSE	 ,					//
		bAlarm5			:= FALSE	,					// 
		bAlarm6			:= FALSE,									//
		bAlarm7			:= FALSE,                                   //
		bAlarm8			:= FALSE,                                   //
		bAlarm9			:= FALSE,                                   //
		bAlarm10		:= FALSE,                                   //
		bAlarm11		:= FALSE,									//
		bAlarm12		:= FALSE,                                   //
		bAlarm13		:= FALSE,                                   //
		bAlarm14		:= FALSE,                                   //
		bAlarm15		:= FALSE,                                   //
		wAlarmCode		=>MesData.MesAlarmCode);
END_METHOD

METHOD M_Init

VAR
	LL	: SINT;
	KK 	: SINT;
	InStruct : ST_ValuesAlarms;
END_VAR
// Create a first alarm after new code activation or PLC restart
//	FIFO.A_Get();
//	FIFO.A_Remove();
	bInit := TRUE;


	GetHostName(bExecute := FALSE);
	GetHostName(bExecute := TRUE);
END_METHOD

END_PROGRAM

// ---- 00_FunctionsBlocks/Beckhoff/Fifo/FB_DBDatasetFifo.TcPOU
FUNCTION_BLOCK FB_DBDatasetFifo
VAR_INPUT
    bOverwrite : BOOL;
    In         : ST_ValuesAlarms;
END_VAR
VAR_OUTPUT
    bOk        : BOOL;
    nCount     : UDINT;
    nLoad      : UDINT;
    Out        : ST_ValuesAlarms;
END_VAR
VAR
    arrBuffer  : ARRAY[0..Max_buffer_size_G] OF BYTE; (* Buffer memory used by FB_MemRingBuffer function block *)
    fbBuffer   : FB_MemRingBuffer;
END_VAR

ACTION A_Add:
fbBuffer.A_AddTail(pWrite := ADR(in),
						   cbWrite:=SIZEOF(in),
						   pBuffer:=ADR(arrBuffer),
						   cbBuffer:=SIZEOF(arrBuffer),
						   bOK=>bOK,
						   nCount =>nCount);
IF NOT bOK THEN 
	IF bOverwrite THEN
		fbBuffer.A_RemoveHead();(*remove one oldest entry*)
		fbBuffer.A_AddTail(bOK => bOk,nCount => nCount);
	END_IF
END_IF

nload := (fbbuffer.cbSize * 100)/(Max_buffer_size_G);
END_ACTION

ACTION A_Get:
fbBuffer.A_GetHead(pWrite := ADR(out),
						   cbWrite:=SIZEOF(out),
						   pBuffer:=ADR(arrBuffer),
						   cbBuffer:=SIZEOF(arrBuffer),
						   bOK=>bOK,
						   nCount =>nCount);
nload := (fbbuffer.cbSize * 100)/(Max_buffer_size_G);
END_ACTION

ACTION A_Remove:
fbBuffer.A_RemoveHead(pRead:=ADR(out),
						cbRead:=SIZEOF(out),
						pBuffer:=ADR(arrBuffer),
						cbBuffer:=SIZEOF(arrBuffer),
						bOK=>bOK,
						nCount =>nCount);
nload := (fbbuffer.cbSize * 100)/(Max_buffer_size_G);
END_ACTION

ACTION A_Reset:
MEMSET(ADR(arrBuffer),0,SIZEOF(arrBuffer)); (*reset internal buffer*)
fbBuffer.A_Reset(bOK=>bOK,nCount=>ncount);
nload := (fbbuffer.cbSize * 100)/(Max_buffer_size_G);
END_ACTION

END_FUNCTION_BLOCK

// ---- 00_FunctionsBlocks/Beckhoff/DataProcessing/WriteFile/FB_WriteFile.TcPOU
FUNCTION_BLOCK FB_WriteFile

VAR_INPUT 
	InDirFile : STRING(1000);
	InAmsId : T_AmsNetID :='';
	InPMessage: POINTER TO BYTE;
	InLMessage: UDINT;
	InStart : BOOL;
	InMode : DWORD := 16#4;	// Append Mode . 
END_VAR

VAR_OUTPUT
	OutBusy 	: BOOL;
	OutError 	: BOOL;
	OutErrorId 	: STRING;
	cbWritten 	: UDINT;
	OutCompleted : BOOL;
END_VAR

VAR 
MesDataExd: LoggerCSV;
	FileHandle 	: UINT;
	select		: INT;
	AX_ErrorId	: ARRAY[1..NbSteps] OF UDINT;
	AX_Error 	: ARRAY[1..NbSteps] OF BOOL;
	OpenFile 	: FB_FileOpen;
	CloseFile 	: FB_FileClose;
	WriteFile 	: FB_FileWrite;
	TextToWrite : STRING(255);
	nSeekPos 	: DINT;
	i 			: UINT;
	bCompleted	: BOOL;
	Trigger		: R_TRIG;
END_VAR

VAR CONSTANT
	NbSteps 	: UINT := 3;
END_VAR

OutCompleted := FALSE;
CASE select OF
	0: // Initialize
		Trigger(CLK := InStart);
		IF Trigger.Q THEN
			select := 1;
			OutBusy := TRUE;
			OutError := FALSE;
			OutErrorId :='';
		END_IF
	1:
		OpenFile(sNetId := InAmsId, 
			sPathName := InDirFile,
			nMode := InMode,
			ePath := Path_generic,
			bExecute := TRUE,
			hFile => FileHandle,
			nErrId => AX_ErrorId[Select],
			bError => AX_Error[Select]
		);
		IF NOT(OpenFile.bBusy) THEN
 			IF NOT(OpenFile.bError) THEN
				select := select+1;
				OpenFile(bExecute := FALSE);
			ELSE
				select := -1;
			END_IF
		END_IF

	2: 
		WriteFile(
			sNetId := InAmsId,
			hFile := FileHandle,
			pWriteBuff := InPMessage,
			cbWriteLen := InLMessage,
			bExecute := TRUE,
			nErrId => AX_ErrorId[Select],
			bError => AX_Error[Select]
		);
		IF NOT(WriteFile.bBusy) THEN
			IF NOT(WriteFile.bError) THEN
				select := select+1;
				WriteFile(bExecute := FALSE);
				cbWritten := WriteFile.cbWrite;
			ELSE
				select := -1;
			END_IF
		END_IF
	3 : 
		CloseFile(sNetId := InAmsId, 
			hFile := FileHandle,
			bExecute := TRUE, 
			tTimeout := T#1S,
			nErrId => AX_ErrorId[Select],
			bError => AX_Error[Select]
		);
		IF NOT(CloseFile.bBusy) THEN
			IF NOT(CloseFile.bError) THEN
				select := 10;
				CloseFile(bExecute := FALSE);
			ELSE
				select := -1;
			END_IF
		END_IF
		
	10: 
		FileHandle := 0;
		OutBusy := FALSE;
		select := 0;
		OutCompleted := TRUE;
		FOR i := 1 TO NbSteps DO
			AX_ErrorId[i] := 0;
			AX_Error[i] := FALSE;
		END_FOR
		
	-1 : 
		IF FileHandle <> 0 THEN
			CloseFile(sNetId := InAmsId, hFile := FileHandle, bExecute := TRUE);
		END_IF
		OpenFile(bExecute := FALSE);
		WriteFile(bExecute := FALSE);
		IF NOT(CloseFIle.bBusy) THEN
			CloseFile(bExecute := FALSE);
		END_IF
		M_AlarmManager();
		select := 10;
END_CASE

METHOD M_AlarmManager : BOOL
VAR
	j : UINT;
	StringInterm : STRING;
END_VAR
OutError := FALSE;
OutErrorId :='';
FOR j := 1 TO NbSteps DO
	OutError := OutError OR AX_Error[j];
	IF AX_Error[j] THEN
		OutErrorId := concat(concat(Concat(UINT_TO_STRING(j),'_'), UDINT_TO_STRING(AX_ERRORID[j])), CONCAT('*',OutErrorId));
	END_IF
END_FOR
END_METHOD

END_FUNCTION_BLOCK

// ---- 00_FunctionsBlocks/Beckhoff/DataProcessing/WriteFile/FUN_CreateDir_CSV.TcPOU
PROGRAM FUN_CreateDir_CSV
VAR_INPUT
	InDirectory 		: T_MaxString;
	Reset2				: BOOL;
END_VAR

VAR
	FB_Time 			: FB_LocalSystemTime;
	MesYear 			: WORD;
	MesMonth			: WORD;
	MesDay				: WORD;
	MesDate				: STRING;
	bTimeOK				: BOOL;
	
	//Dir names 
	CreateDir1			: FB_CreateDir_V2;
	CreateDir2			: FB_CreateDir_V2;
	bFirstDirOk			: BOOL;
	bSecondDirOk		: BOOL;
	bFileOK				: BOOL;
	bDirChange			: BOOL;

END_VAR

VAR_OUTPUT
	
	bInitWrite 			: BOOL;
	AX_DirNames			: ARRAY[1..3] OF t_MaxString; // Folder for years, months and days
	bDirOK				: BOOL;

END_VAR

//	Get time and date  +  Create names
	
IF MesYear <> CalLocalTimeStruct.wYear THEN
	AX_DirNames[1] := Concat(InDirectory, concat(WORD_TO_STRING(CalLocalTimeStruct.wYear), '\'));
	MesYear := CalLocalTimeStruct.wYear;
	bDirChange := TRUE;		
END_IF

IF MesMonth <> CalLocalTimeStruct.wMonth THEN
	AX_DirNames[2] := Concat(AX_DirNames[1], concat(WORD_TO_STRING(CalLocalTimeStruct.wMonth), '\'));
	MesMonth := CalLocalTimeStruct.wMonth;
	bDirChange := TRUE;		
END_IF

IF MesDay <> CalLocalTimeStruct.wDay THEN
	MesDay := CalLocalTimeStruct.wDay;
END_IF		


IF bDirChange OR NOT bFirstDirOk OR NOT bSecondDirOk OR RESET2 THEN
	RESET2 := FALSE;
	bFirstDirOk := FALSE;
	bSecondDirOk := FALSE;
	CreateDir1(InPath := AX_DirNames[1], InExe := TRUE, OutCompleted => bFirstDirOk);
	CreateDir2(InPath := AX_DirNames[2], InExe := bFirstDirOk AND NOT bSecondDirOk, OutCompleted => bSecondDirOk);
	
	IF bFirstDirOk AND bSecondDirOk THEN
		bDirChange := FALSE;
		bDirOK := bFirstDirOk AND bSecondDirOk ;
		CreateDir1(InExe := FALSE);
		CreateDir2(InExe := FALSE);
	END_IF				
END_IF

END_PROGRAM

// ---- 00_FunctionsBlocks/Beckhoff/DataProcessing/WriteFile/FB_CreateDir_V2.TcPOU
FUNCTION_BLOCK FB_CreateDir_V2
VAR_INPUT
	InPath 				: T_Maxstring;
	InExe				: BOOL;
END_VAR
VAR_OUTPUT
	OutExiste			: BOOL;
	OutCompleted		: BOOL;
	OutError			: BOOL;
	OutErrorId			: UDINT;
	OutBusy				: BOOL;
END_VAR
VAR
	CreateDir			: FB_CreateDir;	
	
	Trig_Start			: RS;
	Trig				: R_TRIG;
	
	
END_VAR

Trig(CLK := InExe);
//OutCompleted := NOT Trig.Q AND NOT CreateDir.bBusy AND NOT CreateDir.bError;
Trig_Start(SET := Trig.Q);

CreateDir(
	sNetId := '', 
	sPathName := InPath,
	bExecute := Trig.Q
	);
	
IF Trig_Start.Q1 AND NOT CreateDir.bBusy AND (CreateDir.nErrId = 16#723 OR CreateDir.nErrId = 16#70C ) THEN
	createDir(bExecute := FALSE);
	OutExiste := TRUE;
	OutCompleted := TRUE;
	Trig(CLK := FALSE);
	Trig_Start( RESET1 := OutCompleted OR OutError);
	Trig_Start( RESET1 := FALSE);
ELSIF NOT Trig.Q AND Trig_Start.Q1 AND NOT CreateDir.bBusy AND NOT CreateDir.bError THEN
	OutCompleted := TRUE;
	CreateDir(bExecute := FALSE);
	Trig(CLK := FALSE);
	Trig_Start( RESET1 := OutCompleted OR OutError);
	Trig_Start( RESET1 := FALSE);
ELSIF CreateDir.bError THEN
	OutError := TRUE;
	OutErrorId := CreateDir.nErrid;
	CreateDir(bExecute := FALSE);
	Trig(CLK := FALSE);
	Trig_Start( RESET1 := OutCompleted OR OutError);
	Trig_Start( RESET1 := FALSE);

END_IF

OutBusy := Trig_Start.Q1;

END_FUNCTION_BLOCK

// ---- 00_FunctionsBlocks/Beckhoff/DataProcessing/ReplaceAll.TcPOU
PROGRAM ReplaceAll
// Replaces all the instances of the input string with another string
// If In_StringToSearch := 'aaaaa123aaaaa123aaaaaaa123aaaaa123'
// In_StringToFind := '123'
// In_StringToReplace : = 'ABC'
// Then : OUT_StringToSearch := 'aaaaaABCaaaaaABCaaaaaaaABCaaaaaABC'
// Equivalent to CTRL + H
VAR_INPUT
	IN_StringToSearch	: T_MaxString;		// String to search : main string with instances we wish to replace
	IN_StringToFind		: STRING;			// String we are looking to find in the String_To_Seach
	IN_StringToReplace 	: STRING;			// String with which we want to replace the String To Find in String To Search
END_VAR

VAR_OUTPUT
	OUT_StringToSearch : T_MaxString;		// Output String
END_VAR

VAR
	KK: INT;
	Test_INT : INT;
END_VAR

OUT_StringToSearch := IN_StringToSearch;
FOR KK := 1 TO LEN(STR := OUT_StringToSearch) DO
	Test_INT := FIND(STR1 := OUT_StringToSearch, STR2 := IN_StringToFind);
	IF Test_INT > 0 THEN
		OUT_StringToSearch := REPLACE(STR1 := OUT_StringToSearch, STR2 := IN_StringToReplace, P := Test_INT, L := len(IN_StringToFind));
		KK := Test_Int;
	END_IF
END_FOR

END_PROGRAM

// ---- 04_Application/MAIN/MAIN.TcPOU
PROGRAM MAIN

VAR_INPUT PERSISTENT 
	ParamDisablePLCMaster			: BOOL ;  				(* If true  Force the Redundancy to be on the Slave PLC therefore, no read and write on FB and IO*)
	ParamForceRun					: BOOL ; 				(* Force the PLC to be in run mode .                                *)
	ParamInhibateGridLOC			: BOOL:= FALSE ;			(* Do not switch to slave PLC in case of GRID communication fault   *)
	ParamTest						: BOOL := TRUE ; 		(* If on , do not allow write commands at start up .                *)
	ParamStableOP					: TIME := T#5S ; 
END_VAR

VAR_OUTPUT
	OUT_CalRunningPLC_IO			: BOOL ; 
END_VAR

VAR

	// REDUNDANCY

		TON_Stable 				: TON ;
		FB_MasterBackup			: FB_HeartBeatMasterBackup ;  
 		PLC_ReadSymInfoByName1  : PLC_ReadSymInfoByName	;
		
		CalStableOp_G			: BOOL  ; 

		
	// DATETIME //	
		FB_LocalSystTime      	: FB_LOCALSYSTEMTIME;	// Get time function
		FB_ToGMT : FB_TzSpecificLocalTimeToSystemTime;	// Local to UTC Time function
		TON_Time				: TON;
		CalLocalTimeStruct_Temp: TIMESTRUCT;
		//init
		FB_GetSystemTime        : GETSYSTEMTIME;						// GEt time function
		
		FB_ToLocal 				: FB_FileTimeToTzSpecificLocalTime;		// UTC to local Time function
		fileTime        		: T_FILETIME;							// Filetime format for UTC Time 
		FileTimeLocal			: T_FILETIME;							// Filetime format for local time	

		
	//M_INIT VARIABLE //
		bInit					: BOOL := TRUE ;						// Initialization variable

	R_TRIG_Run: R_TRIG;
	F_TRIG_Run: F_TRIG;

END_VAR

// REDUNDANCY 
	// Heartbit Check
	// Check for ADS variable name every minute. 
	PLC_ReadSymInfoByName1(NETid := CstNetAmsId_Slave, Port:=851,Symname:='MAIN.FB_MasterBackup.nCounter', Start:= CalLocalTimeStruct.wSecond=0 OR bInit,TMOUT:= T#5S) ; 
	FB_MasterBAckup(sNetId:=GVL_CFG.CstNetAmsId_Slave, IdxGroup:=PLC_ReadSymInfoByName1.SYMINFO.idxGroup , IdxOff:=PLC_ReadSymInfoByName1.SYMINFO.idxOffset );

		FB_MasterBAckup.M_Backup() ; 
		FB_MasterBAckup.M_Master() ; 

// INITIALIZATION//
	IF bInit OR CmdInit_G THEN
		M_Init() ; 
		bInit := FALSE; 
	END_IF
	
//GLOBAL VARIABLE UPDATE //
// DateTime 
// Takes some time to query local system time and update the timestamp. 

	TON_Time(IN:= TRUE, PT:=T#1200MS ) ; 
	FB_LocalSystTime(
		bEnable := TRUE,
		dwCycle := 1,
		systemTime => CalLocalTimeStruct_Temp);

	IF TON_Time.Q THEN 
		CalLocalTimeStruct:= CalLocalTimeStruct_Temp ; 
	END_IF
	
	FB_ToGMT(
		in	:= CalLocalTimeStruct,
		tzInfo := CstTimeZone_G,
		out	=> CalGMTTimeStruct);
	
	sTimeGMT_G	:= SYSTEMTIME_TO_STRING(CalGMTTimeStruct);
	sTimeLocal_G	:= SYSTEMTIME_TO_STRING(CalLocalTimeStruct);	

////////// 
// The Master PLC takes cpontrol of the power plant , if it is working and has IEC 104 connection working 
// The Slave PLC takles control if PLC master is not responding or if PLC master does not have IEC 104 working . 
////////// 

TON_Stable( IN:= NOT ParamDisablePLCMaster , PT:= ParamStableOP ) ; // Allow time for the master to read slave data after restart
CalStableOp_G :=  TON_Stable.Q ; 


////////////////////// CODE //////////////////////////////////

// INPUTS //
	PRG_IO.M_Inputs() ;  // Refresh DI and AI 
//	ModbusTcp();	// Update modbus TCP server 

HMI();
	
IF (CstPLCBackup AND (NOT FB_MasterBAckup.bHeartBeat )AND CalStableOp_G) OR (NOT CstPLCBackup AND CalStableOp_G ) OR ParamForceRun  THEN 
// Allow commands, setpoint and orders . 
	OUT_CalRunningPLC_IO := TRUE ; 
// Update redundancy data 
//	Redundancy.M_GetRedundancyData() ; 

ELSIF FB_MasterBAckup.bHeartBeat THEN 
	// Inhib Setpoints and order
	// GET REDUNDANCY DATA FROM DATA 
//	Redundancy.M_ReadRedundancyData() ; 
	OUT_CalRunningPLC_IO := FALSE ; 
ELSE
	
	OUT_CalRunningPLC_IO := FALSE ; 
END_IF 

	A1_PP();

	//PRG_AnnexesFunctions() ; 		// PENSER A DESACTIVER LES ENVOIS DE EMAILS SI REDONDANCE
	//OPC UA 
		OpcUa();
		
// ANALYSIS
	//Analysis();
	
// IO 
	PRG_IO() ; 

// OUTPUTS // 
	PRG_IO.M_Outputs() ;  // Assign DO and AO 

// Database //
	SavePersistent() ;  

//  Au besoin pour inhiber les commandes digitales et les commandes com . 
	R_TRIG_Run(CLK:= OUT_CalRunningPLC_IO) ; 
	F_TRIG_Run(CLK:= OUT_CalRunningPLC_IO) ; 

IF F_TRIG_Run.Q THEN 
	OpcUA.AllDataWPulse.CmdInhibAllWrite 	:= TRUE ; 	// 
	OpcUA.AllDataWPulse.CmdInhibAllRead 	:= TRUE ; 	


ELSIF R_TRIG_Run.Q   THEN 
	IF NOT ParamTest THEN 
		OpcUA.AllDataWPulse.CmdAllowAllWrite	:= TRUE ; 	// Peux ton limiter la réautorization de toutes les ecritures meme si cela avait été forcé à la main auparavant ? 
	END_IF
	OpcUA.AllDataWPulse.CmdAllowAllRead 	:= TRUE ; 	
END_IF

METHOD M_Init : BOOL
VAR_INPUT
END_VAR

VAR 
	Year : STRING ; 
	Month: STRING ; 
	Day : STRING ; 
	Hour: STRING ; 
	Str_Temp: STRING;
END_VAR
//CstCycleTime_G 		:= 50 ;							// Cycle Time
CstTimeZone_G 		:= WEST_EUROPE_TZI ; 		// Local Time Zone 
//Redundancy.M_Init();	



// Get the Windows time ( not accurate ) at startup before updating the system time. 
	// DateTime 
	
	
	FB_GetSystemTime(
		timeLoDW	=> fileTime.dwLowDateTime, 
		timeHiDW	=> fileTime.dwHighDateTime);
		
	FB_ToLocal(
		in			:=fileTime,
		tzInfo 		:= CstTimeZone_G,
		out		 	=> FileTimeLocal);
		
CalLocalTimeStruct := FILETIME_TO_SYSTEMTIME(FileTimelocal) ; 


Year := CONCAT(STR1:= WORD_TO_STRING(CalLocalTimeStruct.wYear), STR2:= '_') ; 
Month := CONCAT(STR1:= WORD_TO_STRING(CalLocalTimeStruct.wMonth), STR2:= '_') ;
Day := CONCAT(STR1:=WORD_TO_STRING(CalLocalTimeStruct.wDay), STR2:= ' ') ;
Hour := CONCAT(STR1:=WORD_TO_STRING(CalLocalTimeStruct.wHour), STR2:= 'h') ;

Str_Temp := Year ; 
Str_Temp := CONCAT(STR1:=Str_Temp , STR2:= Month )  ; 
Str_Temp := CONCAT(STR1:=Str_Temp , STR2:= Day )  ; 	
Str_Temp := CONCAT(STR1:=Str_Temp , STR2:= Hour )  ; 

A1_PP.MesData.MesStartTime 		:= Str_Temp  ; 	// Jour du dernier update de code .
END_METHOD

END_PROGRAM

// ---- 00_FunctionsBlocks/Beckhoff/AlarmManagement/FB_HeartBeatMasterBackup.TcPOU
FUNCTION_BLOCK FB_HeartBeatMasterBackup
//////////////////
// heart beat detector using ADS . 
//////////////////

VAR_INPUT PERSISTENT
	// Parameters of the Object (instance specific) 
	ParamTempoImpulsion3		: TIME := T#500MS ;			// (s) Config : Tempo command impulsion
	ParamTimeout				: TIME  := T#100MS ;				// (Time) Timeout for modbus reading
	                                                    
END_VAR                                                 
                                                        
VAR_INPUT                                               
	//M_Backup Variables//       
//{attribute 'OPC.UA.DA' := '1'}                       
	sNetId 				   		: STRING(20);      					// (NA) ADS device identification Adress
	nPort				  		: UINT := 851;					    // (NA) ADS device Port
	IdxGroup					: UDINT:=16#4020;		// Counter TMC Group Index
	IdxOff						: UDINT:=4; 		// Counter TMC Offset Index
END_VAR                                                             
                                                                    
VAR_OUTPUT                                                          
	bHeartBeat					: BOOL := FALSE;					// (NA) Heart beat detector : False if complete loss of communication with the master
	nCounter                     AT%Q* : BYTE;					    // (NA) Variable to increment in the master	
END_VAR                                                 
                                                        
VAR                                                     
	//M_Backup Variables//                              
	ADSREADEX1                  : ADSREADEX;						// (NA) Functionnal Block to request data from an ADS device
	                                                    			
	TP1							: TP ; 							// (NA) Tempo to define ADS Reading Frequency 
	R_TRIG1						: R_TRIG;							// (NA) Tempo Rising edge detection for ADS Reading
	TON_Freeze					: TON;                                                    			
	ClockRead					: BOOL;								// (NA) ADS reading Clock
	nResult  					: BYTE;            					// (NA) Variable in which the read data have to be stored
	nResult_Temp				: BYTE;	
	bBusy						: BOOL;                             // (NA) Busy Flag
	bError						: BOOL;            					// (NA) Error Flag
	ErrorId						: UDINT;           					// (NA) Error Id returned by FB (see ADS error Code)
	//M_Master Variables//  

	CountError					: UINT ;
	CountOK						: UINT ; 
	
END_VAR

METHOD M_Backup

VAR
	// Method local variables (reinitialized at each cycle) 

END_VAR
TP1(IN:= NOT TP1.Q,PT:=ParamTempoImpulsion3);
R_TRIG1(CLK:=TP1.Q,Q=>ClockRead);

ADSREADEX1(NETID:=sNetId,
		   PORT:=nPort,
		   IDXGRP:=IdxGroup,
		   IDXOFFS:=IdxOff,
		   LEN:=1,
		   READ:=ClockRead,
		   DESTADDR:=ADR(nResult),
		   TMOUT:=ParamTimeout,
		   BUSY=>bBusy,
		   ERR=>bError,
		   ERRID=>ErrorId);
		   

TON_Freeze(IN:= (nResult =nResult_Temp), PT:=ParamTempoImpulsion3 ) ; 		    	   

// Case : after a restart of the master , the Counter  = 0 fixed . Then the slave detects a change 
		   
IF NOT bBusy AND bError THEN
	// IF ADS fails ( Beckhoff is down, not answering ADS) 
	CountError := CountError +1 ; 

ELSIF NOT bBusy AND NOT bError AND NOT TON_Freeze.Q  THEN
	// Return to PLC master OK . OR  Data is incrementing
	CountOK := CountOK+1 ; 
	//bHeartBeat:=TRUE;
	CountError := 0 ; 
	nResult_Temp := nResult ;
ELSIF NOT bBusy AND NOT bError AND TON_Freeze.Q THEN 
	// Counter is frozen ( Master untime stopped , or no stable operation ) 
	bHeartBeat:=FALSE;
	CountError := 0 ; 
	CountOK:= 0 ; 
	nResult_Temp := nResult ;
END_IF


IF CountError > 2  THEN 
	bHeartBeat:=FALSE;
	CountOK:= 0 ; 
ELSIF CountOK>=2 THEN 
	// Return to PLC MAster OK ( makes sure that the change of variables is steady ) 
	bHeartBeat:=TRUE;
END_IF
END_METHOD

METHOD M_Master

VAR
	// Method local variables (reinitialized at each cycle) 
END_VAR
IF MAIN.CalStableOp_G THEN 
	nCounter:=MAX(1,nCounter +1); 			// Return to Master PLC possible . Safe operation
	
ELSE
	
	nCounter:=0;
	
END_IF
END_METHOD

END_FUNCTION_BLOCK

// ---- 04_Application/IO/PRG_IO.TcPOU
PROGRAM PRG_IO
///////////
// This Program is used as an interface between code variable and the I/O cards
//////////
VAR_INPUT
	
//PP States //

// EXECUTE VARIABLES //
	IN_CmdInhibOutput_OPC		: BOOL := TRUE ; 
	MesData				: IO ; 
END_VAR
VAR 	

//M_INIT VARIABLES //
	bInit						: BOOL	:=TRUE ;			// Initialization variables
	iTest                       : INT;
	
	// WAGO Only 
		(*
	xEnable				: 	BOOL := TRUE;
	uiNumberOfModules	: 	UINT;
	xBusy				:	BOOL;
	xError				: 	BOOL;
	sStatus				: 	STRING;
	xKbusInit			: 	BOOL;
	uiNumberOfDO		: 	UINT;
	uiNumberOfDI		: 	UINT;
	uiNumberOfAO		: 	UINT;
	uiNumberOfAI		: 	UINT;
	*)

END_VAR

VAR_INPUT
END_VAR
VAR_INPUT
END_VAR
VAR_INPUT
MesIO_SUBMV_EL1809_1 : ARRAY [1..16] OF ST_DI ; 
MesIO_SUBMV_EL1809_2 : ARRAY [1..16] OF ST_DI ; 
MesIO_SUBMV_EL1809_3 : ARRAY [1..16] OF ST_DI ; 
MesIO_SUBMV_EL2809_4 : ARRAY [1..16] OF ST_DO ; 
MesIO_SUBMV_EL3024_5 : ARRAY [1..4] OF ST_AI ; 
MesIO_PTR_1_EL3024_8 : ARRAY [1..4] OF ST_AI ; 
MesIO_PTR_1_EL1809_9 : ARRAY [1..16] OF ST_DI ; 
MesIO_PTR_1_EL2809_10 : ARRAY [1..16] OF ST_DO ; 
MesIO_PTR_2_EL3024_8 : ARRAY [1..4] OF ST_AI ; 
MesIO_PTR_2_EL1809_9 : ARRAY [1..16] OF ST_DI ; 
MesIO_PTR_2_EL2809_10 : ARRAY [1..16] OF ST_DO ; 
MesIO_PTR_3_EL3024_8 : ARRAY [1..4] OF ST_AI ; 
MesIO_PTR_3_EL1809_9 : ARRAY [1..16] OF ST_DI ; 
MesIO_PTR_3_EL2809_10 : ARRAY [1..16] OF ST_DO ; 
END_VAR

// Initializing the static variables //  
	IF bInit OR CmdInit_G THEN
		M_Init() ; 
		bInit		:= FALSE ; 
		
	END_IF
	M_AlarmManagement() ; 

	(* WAGO Application
	M_Evaluate() ; 
	
	
FR_AppScanKbus.PRG_ScanKbus(
	xEnable				:= xEnable, 
	axDO				:= axDO, 
	aiAO				:= aiAO, 
	axDI				=> axDI, 
	aiAI				=> aiAI, 
	uiNumberOfModules	=> uiNumberOfModules, 
	atypModule			=> atypModule, 
	xBusy				=> xBusy, 
	xError				=> xError, 
	sStatus				=> sStatus, 
	xKbusInit			=> xKbusInit, 
	uiNumberOfDO		=> uiNumberOfDO, 
	uiNumberOfDI		=> uiNumberOfDI, 
	uiNumberOfAO		=> uiNumberOfAO, 
	uiNumberOfAI		=> uiNumberOfAI, 
	tRefresh			:= T#10MS);
	*)

METHOD M_AlarmManagement
//////////////////
// Generates object alarms and manages resets. 
//////////////////

VAR 
	// Method local variables (reinitialized at each cycle) 
	FB_AlarmCodeManager			: FB_AlarmCodeManager ; 

END_VAR

